SPLINE
SPL {X  -165.650, Y  +503.302, Z    +0.000, E1   +50.402, E3 +249333.532}
SPL {X  -165.650, Y  +495.166, Z    +0.000, E1   +51.070, E3 +249343.108}
SPL {X  -165.650, Y  +485.807, Z    +0.000, E1   +51.973, E3 +249352.841}
SPL {X  -165.650, Y  +478.030, Z    +0.000, E1   +52.389, E3 +249362.648}
SPL {X  -165.650, Y  +467.527, Z    +0.000, E1   +53.334, E3 +249373.142}
SPL {X  -165.650, Y  +457.379, Z    +0.000, E1   +53.935, E3 +249384.686}
SPL {X  -165.650, Y  +444.120, Z    +0.000, E1   +54.815, E3 +249398.731}
SPL {X  -165.650, Y  +431.771, Z    +0.000, E1   +55.549, E3 +249411.561}
SPL {X  -165.650, Y  +420.799, Z    +0.000, E1   +56.452, E3 +249420.947}
SPL {X  -165.650, Y  +409.731, Z    +0.000, E1   +57.273, E3 +249430.435}
SPL {X  -165.650, Y  +399.687, Z    +0.000, E1   +57.433, E3 +249442.620}
SPL {X  -165.650, Y  +388.492, Z    +0.000, E1   +57.709, E3 +249455.333}
SPL {X  -165.650, Y  +379.894, Z    +0.000, E1   +57.709, E3 +249466.436}
SPL {X  -165.538, Y  +372.423, Z    +0.000, E1   +57.528, E3 +249477.309}
SPL {X  -164.865, Y  +362.388, Z    +0.000, E1   +57.628, E3 +249489.696}
SPL {X  -163.867, Y  +354.258, Z    +0.000, E1   +57.359, E3 +249501.913}
SPL {X  -162.678, Y  +347.264, Z    +0.000, E1   +57.150, E3 +249512.254}
SPL {X  -161.618, Y  +342.173, Z    +0.000, E1   +56.783, E3 +249521.140}
SPL {X  -159.878, Y  +335.155, Z    +0.000, E1   +56.685, E3 +249530.943}
SPL {X  -158.009, Y  +328.771, Z    +0.000, E1   +56.325, E3 +249541.303}
SPL {X  -156.065, Y  +322.971, Z    +0.000, E1   +56.177, E3 +249549.647}
SPL {X  -154.487, Y  +318.719, Z    +0.000, E1   +55.733, E3 +249557.655}
SPL {X  -151.902, Y  +312.426, Z    +0.000, E1   +55.494, E3 +249567.130}
SPL {X  -149.742, Y  +307.668, Z    +0.000, E1   +54.896, E3 +249576.343}
SPL {X  -146.487, Y  +301.160, Z    +0.000, E1   +54.808, E3 +249585.205}
SPL {X  -133.590, Y  +280.553, Z    +0.000, E1   +59.642, E3 +249586.162}
SPL {X  -112.638, Y  +257.040, Z    +0.000, E1   +51.417, E3 +249689.546}
ENDSPLINE

SPLINE
SPL {X  -115.209, Y  +259.476, Z    +0.000, E1   +49.595, E3 +249722.816}
SPL {X  -147.344, Y  +302.806, Z    +0.000, E1   +40.158, E3 +249812.278}
SPL {X  -160.798, Y  +338.700, Z    +0.000, E1   +25.294, E3 +249811.760}
SPL {X  -163.893, Y  +354.439, Z    +0.000, E1   +16.805, E3 +249806.234}
SPL {X  -165.158, Y  +365.746, Z    +0.000, E1   +10.198, E3 +249804.177}
SPL {X  -165.580, Y  +373.688, Z    +0.000, E1    +5.094, E3 +249803.914}
SPL {X  -165.650, Y  +379.719, Z    +0.000, E1    +0.894, E3 +249803.344}
SPL {X  -165.650, Y  +383.454, Z    +0.000, E1    -2.667, E3 +249802.412}
SPL {X  -165.650, Y  +387.779, Z    +0.000, E1    -8.159, E3 +249802.085}
SPL {X  -165.650, Y  +392.511, Z    +0.000, E1   -14.940, E3 +249800.576}
SPL {X  -165.650, Y  +401.614, Z    +0.000, E1   -27.619, E3 +249801.318}
SPL {X  -165.650, Y  +418.105, Z    +0.000, E1   -49.413, E3 +249796.726}
SPL {X  -165.650, Y  +465.736, Z    +0.000, E1   -65.678, E3 +249810.468}
SPL {X  -165.650, Y  +519.483, Z    +0.000, E1   -68.357, E3 +249836.653}
SPL {X  -165.650, Y  +548.869, Z    +0.000, E1   -62.199, E3 +249892.346}
ENDSPLINE

SPLINE
SPL {X  -165.650, Y  +530.735, Z    +0.000, E1   -57.778, E3 +249900.769}
ENDSPLINE

SPLINE
SPL {X  -165.650, Y  +536.777, Z    +0.000, E1   -57.774, E3 +249908.646}
SPL {X  -165.650, Y  +545.905, Z    +0.000, E1   -57.853, E3 +249919.934}
SPL {X  -165.650, Y  +553.630, Z    +0.000, E1   -57.616, E3 +249931.384}
SPL {X  -165.650, Y  +563.473, Z    +0.000, E1   -57.690, E3 +249943.748}
SPL {X  -165.650, Y  +573.011, Z    +0.000, E1   -57.610, E3 +249956.539}
SPL {X  -165.650, Y  +581.530, Z    +0.000, E1   -57.678, E3 +249967.137}
SPL {X  -165.650, Y  +589.475, Z    +0.000, E1   -57.572, E3 +249978.124}
SPL {X  -165.650, Y  +599.695, Z    +0.000, E1   -57.964, E3 +249988.740}
SPL {X  -165.650, Y  +606.915, Z    +0.000, E1   -57.651, E3 +250000.097}
SPL {X  -165.650, Y  +614.927, Z    +0.000, E1   -57.517, E3 +250011.367}
SPL {X  -165.650, Y  +624.337, Z    +0.000, E1   -57.671, E3 +250022.593}
SPL {X  -165.650, Y  +634.236, Z    +0.000, E1   -57.671, E3 +250035.443}
SPL {X  -165.650, Y  +647.519, Z    +0.000, E1   -57.817, E3 +250051.770}
SPL {X  -165.650, Y  +657.986, Z    +0.000, E1   -57.646, E3 +250066.206}
SPL {X  -165.650, Y  +667.585, Z    +0.000, E1   -57.803, E3 +250077.602}
SPL {X  -165.634, Y  +677.794, Z    +0.000, E1   -57.650, E3 +250091.904}
SPL {X  -165.167, Y  +688.139, Z    +0.000, E1   -57.463, E3 +250106.483}
SPL {X  -164.323, Y  +696.426, Z    +0.000, E1   -57.565, E3 +250116.470}
SPL {X  -163.313, Y  +703.224, Z    +0.000, E1   -57.403, E3 +250126.364}
SPL {X  -161.906, Y  +710.520, Z    +0.000, E1   -57.149, E3 +250137.315}
SPL {X  -160.577, Y  +716.182, Z    +0.000, E1   -56.676, E3 +250147.576}
SPL {X  -158.520, Y  +723.576, Z    +0.000, E1   -56.758, E3 +250156.621}
SPL {X  -156.858, Y  +728.749, Z    +0.000, E1   -56.333, E3 +250165.763}
SPL {X  -155.155, Y  +733.525, Z    +0.000, E1   -55.869, E3 +250174.540}
SPL {X  -153.442, Y  +737.914, Z    +0.000, E1   -55.562, E3 +250181.945}
SPL {X  -150.574, Y  +744.547, Z    +0.000, E1   -55.310, E3 +250191.927}
SPL {X  -147.713, Y  +750.471, Z    +0.000, E1   -54.514, E3 +250203.590}
SPL {X  -139.786, Y  +764.381, Z    +0.000, E1   -57.209, E3 +250207.778}
SPL {X  -110.324, Y  +799.066, Z    +0.000, E1   -54.396, E3 +250276.352}
SPL {X  -100.308, Y  +807.326, Z    +0.000, E1   -52.880, E3 +250320.919}
ENDSPLINE

SPLINE
SPL {X  -108.196, Y  +800.934, Z    +0.000, E1   -52.068, E3 +250413.246}
SPL {X  -144.673, Y  +756.182, Z    +0.000, E1   -41.752, E3 +250431.325}
SPL {X  -160.601, Y  +716.087, Z    +0.000, E1   -25.730, E3 +250430.952}
SPL {X  -164.850, Y  +691.761, Z    +0.000, E1   -12.424, E3 +250428.220}
SPL {X  -165.596, Y  +679.730, Z    +0.000, E1    -4.777, E3 +250427.093}
SPL {X  -165.650, Y  +674.376, Z    +0.000, E1    -0.866, E3 +250427.009}
SPL {X  -165.650, Y  +672.384, Z    +0.000, E1    +0.908, E3 +250425.890}
SPL {X  -165.650, Y  +669.093, Z    +0.000, E1    +4.549, E3 +250425.741}
SPL {X  -165.650, Y  +663.273, Z    +0.000, E1   +12.448, E3 +250424.978}
SPL {X  -165.650, Y  +654.885, Z    +0.000, E1   +25.204, E3 +250423.530}
SPL {X  -165.650, Y  +641.882, Z    +0.000, E1   +46.566, E3 +250416.401}
SPL {X  -165.650, Y  +630.946, Z    +0.000, E1   +55.779, E3 +250417.076}
SPL {X  -165.650, Y  +590.135, Z    +0.000, E1   +59.110, E3 +250449.696}
SPL {X  -165.650, Y  +491.251, Z    +0.000, E1   +65.373, E3 +250509.125}
ENDSPLINE

SPLINE
SPL {X  -165.650, Y  +517.534, Z    +0.000, E1   +59.090, E3 +250523.722}
ENDSPLINE

SPLINE
SPL {X  -165.650, Y  +515.821, Z    +0.000, E1   +58.153, E3 +250532.170}
SPL {X  -165.650, Y  +506.715, Z    +0.000, E1   +58.090, E3 +250544.258}
SPL {X  -165.650, Y  +496.085, Z    +0.000, E1   +57.984, E3 +250558.506}
SPL {X  -165.650, Y  +485.167, Z    +0.000, E1   +58.003, E3 +250572.338}
ENDSPLINE

SPLINE
SPL {X  -165.650, Y  +505.180, Z    +0.000, E1   +52.333, E3 +250579.090}
SPL {X  -165.650, Y  +506.534, Z    +0.000, E1   +50.148, E3 +250590.549}
ENDSPLINE

SPLINE
SPL {X  -165.650, Y  +495.166, Z    +0.000, E1   +51.070, E3 +250603.978}
SPL {X  -165.650, Y  +485.807, Z    +0.000, E1   +51.973, E3 +250613.711}
SPL {X  -165.650, Y  +478.030, Z    +0.000, E1   +52.389, E3 +250623.517}
SPL {X  -165.650, Y  +467.527, Z    +0.000, E1   +53.334, E3 +250634.012}
SPL {X  -165.650, Y  +453.744, Z    +0.000, E1   +54.190, E3 +250649.492}
SPL {X  -165.650, Y  +440.843, Z    +0.000, E1   +55.023, E3 +250662.913}
SPL {X  -165.650, Y  +431.771, Z    +0.000, E1   +55.549, E3 +250672.431}
SPL {X  -165.650, Y  +420.799, Z    +0.000, E1   +56.452, E3 +250681.816}
SPL {X  -165.650, Y  +409.731, Z    +0.000, E1   +57.273, E3 +250691.305}
SPL {X  -165.650, Y  +399.687, Z    +0.000, E1   +57.433, E3 +250703.489}
SPL {X  -165.650, Y  +388.492, Z    +0.000, E1   +57.709, E3 +250716.202}
SPL {X  -165.650, Y  +379.894, Z    +0.000, E1   +57.709, E3 +250727.306}
SPL {X  -165.399, Y  +369.388, Z    +0.000, E1   +57.657, E3 +250741.400}
SPL {X  -164.717, Y  +360.945, Z    +0.000, E1   +57.468, E3 +250753.338}
SPL {X  -163.867, Y  +354.258, Z    +0.000, E1   +57.359, E3 +250762.782}
SPL {X  -162.678, Y  +347.264, Z    +0.000, E1   +57.150, E3 +250773.124}
SPL {X  -161.618, Y  +342.173, Z    +0.000, E1   +56.783, E3 +250782.009}
SPL {X  -159.878, Y  +335.155, Z    +0.000, E1   +56.685, E3 +250791.813}
SPL {X  -158.009, Y  +328.771, Z    +0.000, E1   +56.325, E3 +250802.172}
SPL {X  -156.065, Y  +322.971, Z    +0.000, E1   +56.177, E3 +250810.516}
SPL {X  -153.731, Y  +316.803, Z    +0.000, E1   +55.737, E3 +250821.093}
SPL {X  -150.320, Y  +308.902, Z    +0.000, E1   +55.085, E3 +250834.789}
SPL {X  -147.957, Y  +304.011, Z    +0.000, E1   +54.431, E3 +250844.251}
SPL {X  -144.791, Y  +298.030, Z    +0.000, E1   +55.214, E3 +250848.109}
SPL {X  -133.590, Y  +280.553, Z    +0.000, E1   +59.642, E3 +250847.032}
SPL {X  -112.638, Y  +257.040, Z    +0.000, E1   +51.417, E3 +250950.415}
ENDSPLINE

SPLINE
SPL {X  -115.209, Y  +259.476, Z    +0.000, E1   +49.595, E3 +250983.685}
SPL {X  -147.344, Y  +302.806, Z    +0.000, E1   +40.158, E3 +251073.148}
SPL {X  -160.798, Y  +338.700, Z    +0.000, E1   +25.294, E3 +251072.630}
SPL {X  -163.893, Y  +354.439, Z    +0.000, E1   +16.805, E3 +251067.104}
SPL {X  -165.158, Y  +365.746, Z    +0.000, E1   +10.198, E3 +251065.046}
SPL {X  -165.580, Y  +373.688, Z    +0.000, E1    +5.094, E3 +251064.783}
SPL {X  -165.650, Y  +379.719, Z    +0.000, E1    +0.894, E3 +251064.213}
SPL {X  -165.650, Y  +383.454, Z    +0.000, E1    -2.667, E3 +251063.281}
SPL {X  -165.650, Y  +387.779, Z    +0.000, E1    -8.159, E3 +251062.955}
SPL {X  -165.650, Y  +392.511, Z    +0.000, E1   -14.940, E3 +251061.446}
SPL {X  -165.650, Y  +401.614, Z    +0.000, E1   -27.619, E3 +251062.187}
SPL {X  -165.650, Y  +418.105, Z    +0.000, E1   -49.413, E3 +251057.595}
SPL {X  -165.650, Y  +465.736, Z    +0.000, E1   -65.678, E3 +251071.338}
SPL {X  -165.650, Y  +519.483, Z    +0.000, E1   -68.357, E3 +251097.523}
SPL {X  -165.650, Y  +548.869, Z    +0.000, E1   -62.199, E3 +251153.215}
ENDSPLINE

SPLINE
SPL {X  -165.650, Y  +534.780, Z    +0.000, E1   -57.803, E3 +251166.864}
ENDSPLINE

SPLINE
SPL {X  -165.650, Y  +545.905, Z    +0.000, E1   -57.853, E3 +251180.804}
SPL {X  -165.650, Y  +555.746, Z    +0.000, E1   -57.571, E3 +251195.442}
SPL {X  -165.650, Y  +566.557, Z    +0.000, E1   -57.834, E3 +251207.569}
SPL {X  -165.650, Y  +573.011, Z    +0.000, E1   -57.610, E3 +251217.409}
SPL {X  -165.650, Y  +581.530, Z    +0.000, E1   -57.678, E3 +251228.007}
SPL {X  -165.650, Y  +589.475, Z    +0.000, E1   -57.572, E3 +251238.994}
SPL {X  -165.650, Y  +599.695, Z    +0.000, E1   -57.964, E3 +251249.610}
SPL {X  -165.650, Y  +606.915, Z    +0.000, E1   -57.651, E3 +251260.967}
SPL {X  -165.650, Y  +614.927, Z    +0.000, E1   -57.517, E3 +251272.236}
SPL {X  -165.650, Y  +624.337, Z    +0.000, E1   -57.671, E3 +251283.462}
SPL {X  -165.650, Y  +634.236, Z    +0.000, E1   -57.671, E3 +251296.313}
SPL {X  -165.650, Y  +647.519, Z    +0.000, E1   -57.817, E3 +251312.640}
SPL {X  -165.650, Y  +657.986, Z    +0.000, E1   -57.646, E3 +251327.075}
SPL {X  -165.650, Y  +667.585, Z    +0.000, E1   -57.803, E3 +251338.471}
SPL {X  -165.634, Y  +677.794, Z    +0.000, E1   -57.650, E3 +251352.773}
SPL {X  -165.167, Y  +688.139, Z    +0.000, E1   -57.463, E3 +251367.353}
SPL {X  -164.009, Y  +698.761, Z    +0.000, E1   -57.613, E3 +251380.126}
SPL {X  -162.382, Y  +708.242, Z    +0.000, E1   -57.205, E3 +251395.052}
SPL {X  -160.577, Y  +716.182, Z    +0.000, E1   -56.676, E3 +251408.446}
SPL {X  -158.520, Y  +723.576, Z    +0.000, E1   -56.758, E3 +251417.490}
SPL {X  -156.858, Y  +728.749, Z    +0.000, E1   -56.333, E3 +251426.633}
SPL {X  -155.155, Y  +733.525, Z    +0.000, E1   -55.869, E3 +251435.410}
SPL {X  -152.530, Y  +740.111, Z    +0.000, E1   -55.545, E3 +251445.886}
SPL {X  -149.838, Y  +746.130, Z    +0.000, E1   -55.135, E3 +251455.606}
SPL {X  -147.713, Y  +750.471, Z    +0.000, E1   -54.514, E3 +251464.459}
SPL {X  -139.786, Y  +764.381, Z    +0.000, E1   -57.209, E3 +251468.648}
SPL {X  -110.324, Y  +799.066, Z    +0.000, E1   -54.396, E3 +251537.222}
SPL {X  -100.308, Y  +807.326, Z    +0.000, E1   -52.880, E3 +251581.789}
ENDSPLINE

SPLINE
SPL {X  -108.196, Y  +800.934, Z    +0.000, E1   -52.068, E3 +251674.115}
SPL {X  -147.753, Y  +750.393, Z    +0.000, E1   -39.863, E3 +251692.338}
SPL {X  -161.414, Y  +712.720, Z    +0.000, E1   -24.024, E3 +251691.680}
SPL {X  -164.278, Y  +696.774, Z    +0.000, E1   -15.225, E3 +251686.292}
SPL {X  -165.078, Y  +689.251, Z    +0.000, E1   -10.876, E3 +251690.444}
SPL {X  -165.596, Y  +679.730, Z    +0.000, E1    -4.777, E3 +251687.963}
SPL {X  -165.650, Y  +674.376, Z    +0.000, E1    -0.866, E3 +251687.878}
SPL {X  -165.650, Y  +672.384, Z    +0.000, E1    +0.908, E3 +251686.759}
SPL {X  -165.650, Y  +669.093, Z    +0.000, E1    +4.549, E3 +251686.611}
SPL {X  -165.650, Y  +663.273, Z    +0.000, E1   +12.448, E3 +251685.848}
SPL {X  -165.650, Y  +657.199, Z    +0.000, E1   +21.720, E3 +251685.117}
SPL {X  -165.650, Y  +652.963, Z    +0.000, E1   +28.395, E3 +251683.803}
SPL {X  -165.650, Y  +641.882, Z    +0.000, E1   +46.566, E3 +251677.271}
SPL {X  -165.650, Y  +630.946, Z    +0.000, E1   +55.779, E3 +251677.946}
SPL {X  -165.650, Y  +590.135, Z    +0.000, E1   +59.110, E3 +251710.565}
SPL {X  -165.650, Y  +491.251, Z    +0.000, E1   +65.373, E3 +251769.994}
ENDSPLINE

SPLINE
SPL {X  -165.650, Y  +516.236, Z    +0.000, E1   +58.457, E3 +251790.675}
ENDSPLINE

SPLINE
SPL {X  -165.650, Y  +506.715, Z    +0.000, E1   +58.090, E3 +251805.128}
SPL {X  -165.650, Y  +496.085, Z    +0.000, E1   +57.984, E3 +251819.375}
SPL {X  -165.650, Y  +485.167, Z    +0.000, E1   +58.003, E3 +251833.207}
ENDSPLINE

SPLINE
SPL {X  -165.650, Y  +505.180, Z    +0.000, E1   +52.333, E3 +251839.959}
SPL {X  -165.650, Y  +506.534, Z    +0.000, E1   +50.148, E3 +251851.419}
ENDSPLINE

SPLINE
SPL {X  -165.650, Y  +495.166, Z    +0.000, E1   +51.070, E3 +251864.847}
SPL {X  -165.650, Y  +485.807, Z    +0.000, E1   +51.973, E3 +251874.580}
SPL {X  -165.650, Y  +475.672, Z    +0.000, E1   +52.573, E3 +251887.034}
SPL {X  -165.650, Y  +459.814, Z    +0.000, E1   +53.888, E3 +251903.223}
SPL {X  -165.650, Y  +448.876, Z    +0.000, E1   +54.452, E3 +251915.718}
SPL {X  -165.650, Y  +440.843, Z    +0.000, E1   +55.023, E3 +251923.782}
SPL {X  -165.650, Y  +431.771, Z    +0.000, E1   +55.549, E3 +251933.300}
SPL {X  -165.650, Y  +420.799, Z    +0.000, E1   +56.452, E3 +251942.686}
SPL {X  -165.650, Y  +406.746, Z    +0.000, E1   +57.489, E3 +251954.731}
SPL {X  -165.650, Y  +399.455, Z    +0.000, E1   +57.184, E3 +251966.153}
SPL {X  -165.650, Y  +388.492, Z    +0.000, E1   +57.709, E3 +251977.072}
SPL {X  -165.650, Y  +379.894, Z    +0.000, E1   +57.709, E3 +251988.176}
SPL {X  -165.399, Y  +369.388, Z    +0.000, E1   +57.657, E3 +252002.269}
SPL {X  -164.717, Y  +360.945, Z    +0.000, E1   +57.468, E3 +252014.207}
SPL {X  -163.867, Y  +354.258, Z    +0.000, E1   +57.359, E3 +252023.652}
SPL {X  -162.678, Y  +347.264, Z    +0.000, E1   +57.150, E3 +252033.993}
SPL {X  -160.825, Y  +338.812, Z    +0.000, E1   +56.892, E3 +252046.735}
SPL {X  -158.481, Y  +330.294, Z    +0.000, E1   +56.303, E3 +252061.254}
SPL {X  -156.065, Y  +322.971, Z    +0.000, E1   +56.177, E3 +252071.386}
SPL {X  -154.487, Y  +318.719, Z    +0.000, E1   +55.733, E3 +252079.395}
SPL {X  -151.902, Y  +312.426, Z    +0.000, E1   +55.494, E3 +252088.870}
SPL {X  -148.935, Y  +305.985, Z    +0.000, E1   +54.737, E3 +252101.246}
SPL {X  -144.791, Y  +298.030, Z    +0.000, E1   +55.214, E3 +252108.979}
SPL {X  -133.590, Y  +280.553, Z    +0.000, E1   +59.642, E3 +252107.901}
SPL {X  -112.638, Y  +257.040, Z    +0.000, E1   +51.417, E3 +252211.285}
ENDSPLINE

SPLINE
SPL {X  -115.209, Y  +259.476, Z    +0.000, E1   +49.595, E3 +252244.555}
SPL {X  -147.344, Y  +302.806, Z    +0.000, E1   +40.158, E3 +252334.017}
SPL {X  -160.798, Y  +338.700, Z    +0.000, E1   +25.294, E3 +252333.499}
SPL {X  -163.893, Y  +354.439, Z    +0.000, E1   +16.805, E3 +252327.973}
SPL {X  -165.158, Y  +365.746, Z    +0.000, E1   +10.198, E3 +252325.916}
SPL {X  -165.639, Y  +376.620, Z    +0.000, E1    +3.186, E3 +252325.716}
SPL {X  -165.650, Y  +380.533, Z    +0.000, E1    +0.120, E3 +252324.744}
SPL {X  -165.650, Y  +383.454, Z    +0.000, E1    -2.667, E3 +252324.151}
SPL {X  -165.650, Y  +388.792, Z    +0.000, E1    -9.482, E3 +252323.245}
SPL {X  -165.650, Y  +393.970, Z    +0.000, E1   -17.146, E3 +252322.402}
SPL {X  -165.650, Y  +401.614, Z    +0.000, E1   -27.619, E3 +252323.057}
SPL {X  -165.650, Y  +418.105, Z    +0.000, E1   -49.413, E3 +252318.465}
SPL {X  -165.650, Y  +465.736, Z    +0.000, E1   -65.678, E3 +252332.207}
SPL {X  -165.650, Y  +519.483, Z    +0.000, E1   -68.357, E3 +252358.392}
SPL {X  -165.650, Y  +548.869, Z    +0.000, E1   -62.199, E3 +252414.085}
ENDSPLINE

SPLINE
SPL {X  -165.650, Y  +534.780, Z    +0.000, E1   -57.803, E3 +252427.734}
ENDSPLINE

SPLINE
SPL {X  -165.650, Y  +545.905, Z    +0.000, E1   -57.853, E3 +252441.673}
SPL {X  -165.650, Y  +553.630, Z    +0.000, E1   -57.616, E3 +252453.123}
SPL {X  -165.650, Y  +563.473, Z    +0.000, E1   -57.690, E3 +252465.487}
SPL {X  -165.650, Y  +573.011, Z    +0.000, E1   -57.610, E3 +252478.278}
SPL {X  -165.650, Y  +581.530, Z    +0.000, E1   -57.678, E3 +252488.876}
SPL {X  -165.650, Y  +589.475, Z    +0.000, E1   -57.572, E3 +252499.863}
SPL {X  -165.650, Y  +599.695, Z    +0.000, E1   -57.964, E3 +252510.479}
SPL {X  -165.650, Y  +606.915, Z    +0.000, E1   -57.651, E3 +252521.836}
SPL {X  -165.650, Y  +614.927, Z    +0.000, E1   -57.517, E3 +252533.106}
SPL {X  -165.650, Y  +624.337, Z    +0.000, E1   -57.671, E3 +252544.332}
SPL {X  -165.650, Y  +634.236, Z    +0.000, E1   -57.671, E3 +252557.182}
SPL {X  -165.650, Y  +647.519, Z    +0.000, E1   -57.817, E3 +252573.509}
SPL {X  -165.650, Y  +657.986, Z    +0.000, E1   -57.646, E3 +252587.945}
SPL {X  -165.650, Y  +667.585, Z    +0.000, E1   -57.803, E3 +252599.341}
SPL {X  -165.634, Y  +677.794, Z    +0.000, E1   -57.650, E3 +252613.643}
SPL {X  -165.167, Y  +688.139, Z    +0.000, E1   -57.463, E3 +252628.222}
SPL {X  -164.009, Y  +698.761, Z    +0.000, E1   -57.613, E3 +252640.996}
SPL {X  -162.382, Y  +708.242, Z    +0.000, E1   -57.205, E3 +252655.921}
SPL {X  -160.577, Y  +716.182, Z    +0.000, E1   -56.676, E3 +252669.315}
SPL {X  -158.520, Y  +723.576, Z    +0.000, E1   -56.758, E3 +252678.360}
SPL {X  -156.858, Y  +728.749, Z    +0.000, E1   -56.333, E3 +252687.502}
SPL {X  -155.155, Y  +733.525, Z    +0.000, E1   -55.869, E3 +252696.279}
SPL {X  -153.442, Y  +737.914, Z    +0.000, E1   -55.562, E3 +252703.684}
SPL {X  -150.574, Y  +744.547, Z    +0.000, E1   -55.310, E3 +252713.666}
SPL {X  -147.713, Y  +750.471, Z    +0.000, E1   -54.514, E3 +252725.329}
SPL {X  -139.786, Y  +764.381, Z    +0.000, E1   -57.209, E3 +252729.517}
SPL {X  -110.324, Y  +799.066, Z    +0.000, E1   -54.396, E3 +252798.091}
SPL {X  -100.308, Y  +807.326, Z    +0.000, E1   -52.880, E3 +252842.658}
ENDSPLINE

SPLINE
SPL {X  -108.196, Y  +800.934, Z    +0.000, E1   -52.068, E3 +252934.985}
SPL {X  -144.673, Y  +756.182, Z    +0.000, E1   -41.752, E3 +252953.064}
SPL {X  -160.601, Y  +716.087, Z    +0.000, E1   -25.730, E3 +252952.691}
SPL {X  -164.850, Y  +691.761, Z    +0.000, E1   -12.424, E3 +252949.959}
SPL {X  -165.596, Y  +679.730, Z    +0.000, E1    -4.777, E3 +252948.832}
SPL {X  -165.650, Y  +674.376, Z    +0.000, E1    -0.866, E3 +252948.748}
SPL {X  -165.650, Y  +672.384, Z    +0.000, E1    +0.908, E3 +252947.629}
SPL {X  -165.650, Y  +669.093, Z    +0.000, E1    +4.549, E3 +252947.480}
SPL {X  -165.650, Y  +663.273, Z    +0.000, E1   +12.448, E3 +252946.717}
SPL {X  -165.650, Y  +654.885, Z    +0.000, E1   +25.204, E3 +252945.269}
SPL {X  -165.650, Y  +641.882, Z    +0.000, E1   +46.566, E3 +252938.140}
SPL {X  -165.650, Y  +630.946, Z    +0.000, E1   +55.779, E3 +252938.815}
SPL {X  -165.650, Y  +595.858, Z    +0.000, E1   +64.262, E3 +252953.696}
SPL {X  -165.650, Y  +589.368, Z    +0.000, E1   +58.232, E3 +252974.437}
SPL {X  -165.650, Y  +491.251, Z    +0.000, E1   +65.373, E3 +253030.864}
ENDSPLINE

SPLINE
SPL {X  -165.650, Y  +516.236, Z    +0.000, E1   +58.457, E3 +253051.545}
ENDSPLINE

SPLINE
SPL {X  -165.650, Y  +506.715, Z    +0.000, E1   +58.090, E3 +253065.998}
SPL {X  -165.650, Y  +496.085, Z    +0.000, E1   +57.984, E3 +253080.245}
SPL {X  -165.650, Y  +485.167, Z    +0.000, E1   +58.003, E3 +253094.077}
ENDSPLINE

SPLINE
SPL {X  -165.650, Y  +505.180, Z    +0.000, E1   +52.333, E3 +253100.829}
SPL {X  -165.650, Y  +506.534, Z    +0.000, E1   +50.148, E3 +253112.288}
ENDSPLINE

SPLINE
SPL {X  -165.650, Y  +495.166, Z    +0.000, E1   +51.070, E3 +253125.717}
SPL {X  -165.650, Y  +485.807, Z    +0.000, E1   +51.973, E3 +253135.450}
SPL {X  -165.650, Y  +475.672, Z    +0.000, E1   +52.573, E3 +253147.903}
SPL {X  -165.650, Y  +459.814, Z    +0.000, E1   +53.888, E3 +253164.093}
SPL {X  -165.650, Y  +448.876, Z    +0.000, E1   +54.452, E3 +253176.588}
SPL {X  -165.650, Y  +440.843, Z    +0.000, E1   +55.023, E3 +253184.652}
SPL {X  -165.650, Y  +431.771, Z    +0.000, E1   +55.549, E3 +253194.170}
SPL {X  -165.650, Y  +420.799, Z    +0.000, E1   +56.452, E3 +253203.555}
SPL {X  -165.650, Y  +409.731, Z    +0.000, E1   +57.273, E3 +253213.044}
SPL {X  -165.650, Y  +399.687, Z    +0.000, E1   +57.433, E3 +253225.228}
SPL {X  -165.650, Y  +388.492, Z    +0.000, E1   +57.709, E3 +253237.941}
SPL {X  -165.650, Y  +379.894, Z    +0.000, E1   +57.709, E3 +253249.045}
SPL {X  -165.538, Y  +372.423, Z    +0.000, E1   +57.528, E3 +253259.918}
SPL {X  -164.865, Y  +362.388, Z    +0.000, E1   +57.628, E3 +253272.305}
SPL {X  -163.867, Y  +354.258, Z    +0.000, E1   +57.359, E3 +253284.521}
SPL {X  -162.678, Y  +347.264, Z    +0.000, E1   +57.150, E3 +253294.863}
SPL {X  -161.618, Y  +342.173, Z    +0.000, E1   +56.783, E3 +253303.748}
SPL {X  -159.878, Y  +335.155, Z    +0.000, E1   +56.685, E3 +253313.552}
SPL {X  -158.009, Y  +328.771, Z    +0.000, E1   +56.325, E3 +253323.912}
SPL {X  -156.065, Y  +322.971, Z    +0.000, E1   +56.177, E3 +253332.256}
SPL {X  -154.487, Y  +318.719, Z    +0.000, E1   +55.733, E3 +253340.264}
SPL {X  -151.902, Y  +312.426, Z    +0.000, E1   +55.494, E3 +253349.739}
SPL {X  -148.935, Y  +305.985, Z    +0.000, E1   +54.737, E3 +253362.116}
SPL {X  -144.791, Y  +298.030, Z    +0.000, E1   +55.214, E3 +253369.848}
SPL {X  -133.590, Y  +280.553, Z    +0.000, E1   +59.642, E3 +253368.771}
SPL {X  -112.638, Y  +257.040, Z    +0.000, E1   +51.417, E3 +253472.154}
ENDSPLINE

SPLINE
SPL {X  -115.209, Y  +259.476, Z    +0.000, E1   +49.595, E3 +253505.425}
SPL {X  -147.344, Y  +302.806, Z    +0.000, E1   +40.158, E3 +253594.887}
SPL {X  -160.798, Y  +338.700, Z    +0.000, E1   +25.294, E3 +253594.369}
SPL {X  -163.893, Y  +354.439, Z    +0.000, E1   +16.805, E3 +253588.843}
SPL {X  -165.158, Y  +365.746, Z    +0.000, E1   +10.198, E3 +253586.786}
SPL {X  -165.580, Y  +373.688, Z    +0.000, E1    +5.094, E3 +253586.523}
SPL {X  -165.650, Y  +378.140, Z    +0.000, E1    +1.996, E3 +253586.609}
SPL {X  -165.650, Y  +381.477, Z    +0.000, E1    -0.622, E3 +253585.396}
SPL {X  -165.650, Y  +384.861, Z    +0.000, E1    -4.465, E3 +253584.799}
SPL {X  -165.650, Y  +388.792, Z    +0.000, E1    -9.482, E3 +253584.115}
SPL {X  -165.650, Y  +393.970, Z    +0.000, E1   -17.146, E3 +253583.271}
SPL {X  -165.650, Y  +401.614, Z    +0.000, E1   -27.619, E3 +253583.926}
SPL {X  -165.650, Y  +418.105, Z    +0.000, E1   -49.413, E3 +253579.334}
SPL {X  -165.650, Y  +465.736, Z    +0.000, E1   -65.678, E3 +253593.077}
SPL {X  -165.650, Y  +519.483, Z    +0.000, E1   -68.357, E3 +253619.262}
SPL {X  -165.650, Y  +548.869, Z    +0.000, E1   -62.199, E3 +253674.954}
ENDSPLINE

SPLINE
SPL {X  -165.650, Y  +534.780, Z    +0.000, E1   -57.803, E3 +253688.604}
ENDSPLINE

SPLINE
SPL {X  -165.650, Y  +545.905, Z    +0.000, E1   -57.853, E3 +253702.543}
SPL {X  -165.650, Y  +553.630, Z    +0.000, E1   -57.616, E3 +253713.993}
SPL {X  -165.650, Y  +563.473, Z    +0.000, E1   -57.690, E3 +253726.357}
SPL {X  -165.650, Y  +573.011, Z    +0.000, E1   -57.610, E3 +253739.148}
SPL {X  -165.650, Y  +581.530, Z    +0.000, E1   -57.678, E3 +253749.746}
SPL {X  -165.650, Y  +589.475, Z    +0.000, E1   -57.572, E3 +253760.733}
SPL {X  -165.650, Y  +599.695, Z    +0.000, E1   -57.964, E3 +253771.349}
SPL {X  -165.650, Y  +606.915, Z    +0.000, E1   -57.651, E3 +253782.706}
SPL {X  -165.650, Y  +614.927, Z    +0.000, E1   -57.517, E3 +253793.975}
SPL {X  -165.650, Y  +624.337, Z    +0.000, E1   -57.671, E3 +253805.201}
SPL {X  -165.650, Y  +634.236, Z    +0.000, E1   -57.671, E3 +253818.052}
SPL {X  -165.650, Y  +647.519, Z    +0.000, E1   -57.817, E3 +253834.379}
SPL {X  -165.650, Y  +657.986, Z    +0.000, E1   -57.646, E3 +253848.814}
SPL {X  -165.650, Y  +667.585, Z    +0.000, E1   -57.803, E3 +253860.210}
SPL {X  -165.634, Y  +677.794, Z    +0.000, E1   -57.650, E3 +253874.512}
SPL {X  -165.167, Y  +688.139, Z    +0.000, E1   -57.463, E3 +253889.092}
SPL {X  -164.009, Y  +698.761, Z    +0.000, E1   -57.613, E3 +253901.865}
SPL {X  -162.382, Y  +708.242, Z    +0.000, E1   -57.205, E3 +253916.791}
SPL {X  -160.577, Y  +716.182, Z    +0.000, E1   -56.676, E3 +253930.185}
SPL {X  -158.520, Y  +723.576, Z    +0.000, E1   -56.758, E3 +253939.230}
SPL {X  -156.858, Y  +728.749, Z    +0.000, E1   -56.333, E3 +253948.372}
SPL {X  -155.155, Y  +733.525, Z    +0.000, E1   -55.869, E3 +253957.149}
SPL {X  -152.530, Y  +740.111, Z    +0.000, E1   -55.545, E3 +253967.625}
SPL {X  -149.838, Y  +746.130, Z    +0.000, E1   -55.135, E3 +253977.345}
SPL {X  -147.713, Y  +750.471, Z    +0.000, E1   -54.514, E3 +253986.199}
SPL {X  -139.786, Y  +764.381, Z    +0.000, E1   -57.209, E3 +253990.387}
SPL {X  -110.324, Y  +799.066, Z    +0.000, E1   -54.396, E3 +254058.961}
SPL {X  -100.308, Y  +807.326, Z    +0.000, E1   -52.880, E3 +254103.528}
ENDSPLINE

SPLINE
SPL {X  -108.196, Y  +800.934, Z    +0.000, E1   -52.068, E3 +254195.854}
SPL {X  -144.673, Y  +756.182, Z    +0.000, E1   -41.752, E3 +254213.933}
SPL {X  -160.601, Y  +716.087, Z    +0.000, E1   -25.730, E3 +254213.561}
SPL {X  -164.850, Y  +691.761, Z    +0.000, E1   -12.424, E3 +254210.828}
SPL {X  -165.596, Y  +679.730, Z    +0.000, E1    -4.777, E3 +254209.702}
SPL {X  -165.650, Y  +674.376, Z    +0.000, E1    -0.866, E3 +254209.617}
SPL {X  -165.650, Y  +672.384, Z    +0.000, E1    +0.908, E3 +254208.498}
SPL {X  -165.650, Y  +669.968, Z    +0.000, E1    +3.584, E3 +254208.314}
SPL {X  -165.650, Y  +666.667, Z    +0.000, E1    +7.761, E3 +254207.993}
SPL {X  -165.650, Y  +662.028, Z    +0.000, E1   +14.359, E3 +254207.624}
SPL {X  -165.650, Y  +654.885, Z    +0.000, E1   +25.204, E3 +254206.139}
SPL {X  -165.650, Y  +641.882, Z    +0.000, E1   +46.566, E3 +254199.010}
SPL {X  -165.650, Y  +630.946, Z    +0.000, E1   +55.779, E3 +254199.685}
SPL {X  -165.650, Y  +590.135, Z    +0.000, E1   +59.110, E3 +254232.304}
SPL {X  -165.650, Y  +491.251, Z    +0.000, E1   +65.373, E3 +254291.734}
ENDSPLINE

SPLINE
SPL {X  -165.650, Y  +516.236, Z    +0.000, E1   +58.457, E3 +254312.414}
ENDSPLINE

SPLINE
SPL {X  -165.650, Y  +506.715, Z    +0.000, E1   +58.090, E3 +254326.867}
SPL {X  -165.650, Y  +496.085, Z    +0.000, E1   +57.984, E3 +254341.115}
SPL {X  -165.650, Y  +485.167, Z    +0.000, E1   +58.003, E3 +254354.946}
ENDSPLINE

SPLINE
SPL {X  -165.650, Y  +505.180, Z    +0.000, E1   +52.333, E3 +254361.698}
SPL {X  -165.650, Y  +506.534, Z    +0.000, E1   +50.148, E3 +254373.158}
ENDSPLINE

SPLINE
SPL {X  -165.650, Y  +495.166, Z    +0.000, E1   +51.070, E3 +254386.586}
SPL {X  -165.650, Y  +485.807, Z    +0.000, E1   +51.973, E3 +254396.319}
SPL {X  -165.650, Y  +478.030, Z    +0.000, E1   +52.389, E3 +254406.126}
SPL {X  -165.650, Y  +467.527, Z    +0.000, E1   +53.334, E3 +254416.620}
SPL {X  -165.650, Y  +457.379, Z    +0.000, E1   +53.935, E3 +254428.164}
SPL {X  -165.650, Y  +444.120, Z    +0.000, E1   +54.815, E3 +254442.209}
SPL {X  -165.650, Y  +431.771, Z    +0.000, E1   +55.549, E3 +254455.039}
SPL {X  -165.650, Y  +420.799, Z    +0.000, E1   +56.452, E3 +254464.425}
SPL {X  -165.650, Y  +409.731, Z    +0.000, E1   +57.273, E3 +254473.913}
SPL {X  -165.650, Y  +399.687, Z    +0.000, E1   +57.433, E3 +254486.098}
SPL {X  -165.650, Y  +388.492, Z    +0.000, E1   +57.709, E3 +254498.811}
SPL {X  -165.650, Y  +379.894, Z    +0.000, E1   +57.709, E3 +254509.915}
SPL {X  -165.538, Y  +372.423, Z    +0.000, E1   +57.528, E3 +254520.788}
SPL {X  -164.865, Y  +362.388, Z    +0.000, E1   +57.628, E3 +254533.174}
SPL {X  -163.867, Y  +354.258, Z    +0.000, E1   +57.359, E3 +254545.391}
SPL {X  -162.678, Y  +347.264, Z    +0.000, E1   +57.150, E3 +254555.732}
SPL {X  -161.618, Y  +342.173, Z    +0.000, E1   +56.783, E3 +254564.618}
SPL {X  -159.878, Y  +335.155, Z    +0.000, E1   +56.685, E3 +254574.421}
SPL {X  -158.009, Y  +328.771, Z    +0.000, E1   +56.325, E3 +254584.781}
SPL {X  -156.065, Y  +322.971, Z    +0.000, E1   +56.177, E3 +254593.125}
SPL {X  -154.487, Y  +318.719, Z    +0.000, E1   +55.733, E3 +254601.134}
SPL {X  -151.902, Y  +312.426, Z    +0.000, E1   +55.494, E3 +254610.609}
SPL {X  -149.742, Y  +307.668, Z    +0.000, E1   +54.896, E3 +254619.821}
SPL {X  -146.487, Y  +301.160, Z    +0.000, E1   +54.808, E3 +254628.684}
SPL {X  -133.590, Y  +280.553, Z    +0.000, E1   +59.642, E3 +254629.641}
SPL {X  -112.638, Y  +257.040, Z    +0.000, E1   +51.417, E3 +254733.024}
ENDSPLINE

SPLINE
SPL {X  -115.209, Y  +259.476, Z    +0.000, E1   +49.595, E3 +254766.294}
SPL {X  -147.344, Y  +302.806, Z    +0.000, E1   +40.158, E3 +254855.756}
SPL {X  -160.798, Y  +338.700, Z    +0.000, E1   +25.294, E3 +254855.238}
SPL {X  -163.893, Y  +354.439, Z    +0.000, E1   +16.805, E3 +254849.712}
SPL {X  -165.158, Y  +365.746, Z    +0.000, E1   +10.198, E3 +254847.655}
SPL {X  -165.639, Y  +376.620, Z    +0.000, E1    +3.186, E3 +254847.455}
SPL {X  -165.650, Y  +381.477, Z    +0.000, E1    -0.622, E3 +254846.266}
SPL {X  -165.650, Y  +386.363, Z    +0.000, E1    -6.162, E3 +254845.614}
SPL {X  -165.650, Y  +392.511, Z    +0.000, E1   -14.940, E3 +254844.054}
SPL {X  -165.650, Y  +398.939, Z    +0.000, E1   -23.851, E3 +254845.439}
SPL {X  -165.650, Y  +404.249, Z    +0.000, E1   -31.650, E3 +254844.161}
SPL {X  -165.650, Y  +418.105, Z    +0.000, E1   -49.413, E3 +254840.204}
SPL {X  -165.650, Y  +465.736, Z    +0.000, E1   -65.678, E3 +254853.946}
SPL {X  -165.650, Y  +519.483, Z    +0.000, E1   -68.357, E3 +254880.131}
SPL {X  -165.650, Y  +548.869, Z    +0.000, E1   -62.199, E3 +254935.824}
ENDSPLINE

SPLINE
SPL {X  -165.650, Y  +530.735, Z    +0.000, E1   -57.778, E3 +254944.247}
ENDSPLINE

SPLINE
SPL {X  -165.650, Y  +536.777, Z    +0.000, E1   -57.774, E3 +254952.124}
SPL {X  -165.650, Y  +545.905, Z    +0.000, E1   -57.853, E3 +254963.413}
SPL {X  -165.650, Y  +553.630, Z    +0.000, E1   -57.616, E3 +254974.862}
SPL {X  -165.650, Y  +563.473, Z    +0.000, E1   -57.690, E3 +254987.226}
SPL {X  -165.650, Y  +573.011, Z    +0.000, E1   -57.610, E3 +255000.017}
SPL {X  -165.650, Y  +581.530, Z    +0.000, E1   -57.678, E3 +255010.615}
SPL {X  -165.650, Y  +589.475, Z    +0.000, E1   -57.572, E3 +255021.602}
SPL {X  -165.650, Y  +599.695, Z    +0.000, E1   -57.964, E3 +255032.218}
SPL {X  -165.650, Y  +606.915, Z    +0.000, E1   -57.651, E3 +255043.575}
SPL {X  -165.650, Y  +614.927, Z    +0.000, E1   -57.517, E3 +255054.845}
SPL {X  -165.650, Y  +624.337, Z    +0.000, E1   -57.671, E3 +255066.071}
SPL {X  -165.650, Y  +634.236, Z    +0.000, E1   -57.671, E3 +255078.921}
SPL {X  -165.650, Y  +647.519, Z    +0.000, E1   -57.817, E3 +255095.249}
SPL {X  -165.650, Y  +657.986, Z    +0.000, E1   -57.646, E3 +255109.684}
SPL {X  -165.650, Y  +667.585, Z    +0.000, E1   -57.803, E3 +255121.080}
SPL {X  -165.634, Y  +677.794, Z    +0.000, E1   -57.650, E3 +255135.382}
SPL {X  -165.167, Y  +688.139, Z    +0.000, E1   -57.463, E3 +255149.961}
SPL {X  -164.323, Y  +696.426, Z    +0.000, E1   -57.565, E3 +255159.948}
SPL {X  -163.313, Y  +703.224, Z    +0.000, E1   -57.403, E3 +255169.842}
SPL {X  -161.906, Y  +710.520, Z    +0.000, E1   -57.149, E3 +255180.793}
SPL {X  -160.577, Y  +716.182, Z    +0.000, E1   -56.676, E3 +255191.054}
SPL {X  -158.520, Y  +723.576, Z    +0.000, E1   -56.758, E3 +255200.099}
SPL {X  -156.858, Y  +728.749, Z    +0.000, E1   -56.333, E3 +255209.242}
SPL {X  -155.155, Y  +733.525, Z    +0.000, E1   -55.869, E3 +255218.018}
SPL {X  -153.442, Y  +737.914, Z    +0.000, E1   -55.562, E3 +255225.423}
SPL {X  -150.574, Y  +744.547, Z    +0.000, E1   -55.310, E3 +255235.405}
SPL {X  -147.713, Y  +750.471, Z    +0.000, E1   -54.514, E3 +255247.068}
SPL {X  -139.786, Y  +764.381, Z    +0.000, E1   -57.209, E3 +255251.256}
SPL {X  -110.324, Y  +799.066, Z    +0.000, E1   -54.396, E3 +255319.830}
SPL {X  -100.308, Y  +807.326, Z    +0.000, E1   -52.880, E3 +255364.398}
ENDSPLINE

SPLINE
SPL {X  -108.196, Y  +800.934, Z    +0.000, E1   -52.068, E3 +255456.724}
SPL {X  -144.673, Y  +756.182, Z    +0.000, E1   -41.752, E3 +255474.803}
SPL {X  -160.601, Y  +716.087, Z    +0.000, E1   -25.730, E3 +255474.430}
SPL {X  -164.850, Y  +691.761, Z    +0.000, E1   -12.424, E3 +255471.698}
SPL {X  -165.596, Y  +679.730, Z    +0.000, E1    -4.777, E3 +255470.572}
SPL {X  -165.650, Y  +674.376, Z    +0.000, E1    -0.866, E3 +255470.487}
SPL {X  -165.650, Y  +672.384, Z    +0.000, E1    +0.908, E3 +255469.368}
SPL {X  -165.650, Y  +669.093, Z    +0.000, E1    +4.549, E3 +255469.219}
SPL {X  -165.650, Y  +663.273, Z    +0.000, E1   +12.448, E3 +255468.457}
SPL {X  -165.650, Y  +654.885, Z    +0.000, E1   +25.204, E3 +255467.008}
SPL {X  -165.650, Y  +641.882, Z    +0.000, E1   +46.566, E3 +255459.880}
SPL {X  -165.650, Y  +630.946, Z    +0.000, E1   +55.779, E3 +255460.554}
SPL {X  -165.650, Y  +590.135, Z    +0.000, E1   +59.110, E3 +255493.174}
SPL {X  -165.650, Y  +491.251, Z    +0.000, E1   +65.373, E3 +255552.603}
ENDSPLINE

SPLINE
SPL {X  -165.650, Y  +517.534, Z    +0.000, E1   +59.090, E3 +255567.201}
ENDSPLINE

SPLINE
SPL {X  -165.650, Y  +515.821, Z    +0.000, E1   +58.153, E3 +255575.648}
SPL {X  -165.650, Y  +506.715, Z    +0.000, E1   +58.090, E3 +255587.737}
SPL {X  -165.650, Y  +496.085, Z    +0.000, E1   +57.984, E3 +255601.984}
SPL {X  -165.650, Y  +485.167, Z    +0.000, E1   +58.003, E3 +255615.816}
ENDSPLINE

SPLINE
SPL {X  -165.650, Y  +505.180, Z    +0.000, E1   +52.333, E3 +255622.568}
SPL {X  -165.650, Y  +506.534, Z    +0.000, E1   +50.148, E3 +255634.028}
ENDSPLINE

SPLINE
SPL {X  -165.650, Y  +495.166, Z    +0.000, E1   +51.070, E3 +255647.456}
SPL {X  -165.650, Y  +485.807, Z    +0.000, E1   +51.973, E3 +255657.189}
SPL {X  -165.650, Y  +478.030, Z    +0.000, E1   +52.389, E3 +255666.996}
SPL {X  -165.650, Y  +467.527, Z    +0.000, E1   +53.334, E3 +255677.490}
SPL {X  -165.650, Y  +453.744, Z    +0.000, E1   +54.190, E3 +255692.971}
SPL {X  -165.650, Y  +440.843, Z    +0.000, E1   +55.023, E3 +255706.391}
SPL {X  -165.650, Y  +431.771, Z    +0.000, E1   +55.549, E3 +255715.909}
SPL {X  -165.650, Y  +420.799, Z    +0.000, E1   +56.452, E3 +255725.295}
SPL {X  -165.650, Y  +409.731, Z    +0.000, E1   +57.273, E3 +255734.783}
SPL {X  -165.650, Y  +399.687, Z    +0.000, E1   +57.433, E3 +255746.967}
SPL {X  -165.650, Y  +388.492, Z    +0.000, E1   +57.709, E3 +255759.681}
SPL {X  -165.650, Y  +379.894, Z    +0.000, E1   +57.709, E3 +255770.784}
SPL {X  -165.399, Y  +369.388, Z    +0.000, E1   +57.657, E3 +255784.878}
SPL {X  -164.717, Y  +360.945, Z    +0.000, E1   +57.468, E3 +255796.816}
SPL {X  -163.867, Y  +354.258, Z    +0.000, E1   +57.359, E3 +255806.261}
SPL {X  -162.678, Y  +347.264, Z    +0.000, E1   +57.150, E3 +255816.602}
SPL {X  -161.618, Y  +342.173, Z    +0.000, E1   +56.783, E3 +255825.487}
SPL {X  -159.878, Y  +335.155, Z    +0.000, E1   +56.685, E3 +255835.291}
SPL {X  -158.009, Y  +328.771, Z    +0.000, E1   +56.325, E3 +255845.651}
SPL {X  -156.065, Y  +322.971, Z    +0.000, E1   +56.177, E3 +255853.995}
SPL {X  -153.731, Y  +316.803, Z    +0.000, E1   +55.737, E3 +255864.571}
SPL {X  -150.320, Y  +308.902, Z    +0.000, E1   +55.085, E3 +255878.267}
SPL {X  -147.957, Y  +304.011, Z    +0.000, E1   +54.431, E3 +255887.730}
SPL {X  -144.791, Y  +298.030, Z    +0.000, E1   +55.214, E3 +255891.587}
SPL {X  -133.590, Y  +280.553, Z    +0.000, E1   +59.642, E3 +255890.510}
SPL {X  -112.638, Y  +257.040, Z    +0.000, E1   +51.417, E3 +255993.893}
ENDSPLINE

SPLINE
SPL {X  -115.209, Y  +259.476, Z    +0.000, E1   +49.595, E3 +256027.164}
SPL {X  -147.344, Y  +302.806, Z    +0.000, E1   +40.158, E3 +256116.626}
SPL {X  -160.798, Y  +338.700, Z    +0.000, E1   +25.294, E3 +256116.108}
SPL {X  -163.893, Y  +354.439, Z    +0.000, E1   +16.805, E3 +256110.582}
SPL {X  -165.158, Y  +365.746, Z    +0.000, E1   +10.198, E3 +256108.525}
SPL {X  -165.580, Y  +373.688, Z    +0.000, E1    +5.094, E3 +256108.262}
SPL {X  -165.650, Y  +379.719, Z    +0.000, E1    +0.894, E3 +256107.692}
SPL {X  -165.650, Y  +383.454, Z    +0.000, E1    -2.667, E3 +256106.760}
SPL {X  -165.650, Y  +387.779, Z    +0.000, E1    -8.159, E3 +256106.433}
SPL {X  -165.650, Y  +392.511, Z    +0.000, E1   -14.940, E3 +256104.924}
SPL {X  -165.650, Y  +401.614, Z    +0.000, E1   -27.619, E3 +256105.666}
SPL {X  -165.650, Y  +418.105, Z    +0.000, E1   -49.413, E3 +256101.073}
SPL {X  -165.650, Y  +465.736, Z    +0.000, E1   -65.678, E3 +256114.816}
SPL {X  -165.650, Y  +519.483, Z    +0.000, E1   -68.357, E3 +256141.001}
SPL {X  -165.650, Y  +548.869, Z    +0.000, E1   -62.199, E3 +256196.693}
ENDSPLINE

SPLINE
SPL {X  -165.650, Y  +534.780, Z    +0.000, E1   -57.803, E3 +256210.343}
ENDSPLINE

SPLINE
SPL {X  -165.650, Y  +545.905, Z    +0.000, E1   -57.853, E3 +256224.282}
SPL {X  -165.650, Y  +555.746, Z    +0.000, E1   -57.571, E3 +256238.920}
SPL {X  -165.650, Y  +566.557, Z    +0.000, E1   -57.834, E3 +256251.048}
SPL {X  -165.650, Y  +573.011, Z    +0.000, E1   -57.610, E3 +256260.887}
SPL {X  -165.650, Y  +581.530, Z    +0.000, E1   -57.678, E3 +256271.485}
SPL {X  -165.650, Y  +589.475, Z    +0.000, E1   -57.572, E3 +256282.472}
SPL {X  -165.650, Y  +599.695, Z    +0.000, E1   -57.964, E3 +256293.088}
SPL {X  -165.650, Y  +606.915, Z    +0.000, E1   -57.651, E3 +256304.445}
SPL {X  -165.650, Y  +614.927, Z    +0.000, E1   -57.517, E3 +256315.715}
SPL {X  -165.650, Y  +624.337, Z    +0.000, E1   -57.671, E3 +256326.940}
SPL {X  -165.650, Y  +634.236, Z    +0.000, E1   -57.671, E3 +256339.791}
SPL {X  -165.650, Y  +647.519, Z    +0.000, E1   -57.817, E3 +256356.118}
SPL {X  -165.650, Y  +657.986, Z    +0.000, E1   -57.646, E3 +256370.554}
SPL {X  -165.650, Y  +667.585, Z    +0.000, E1   -57.803, E3 +256381.949}
SPL {X  -165.634, Y  +677.794, Z    +0.000, E1   -57.650, E3 +256396.252}
SPL {X  -165.167, Y  +688.139, Z    +0.000, E1   -57.463, E3 +256410.831}
SPL {X  -164.009, Y  +698.761, Z    +0.000, E1   -57.613, E3 +256423.604}
SPL {X  -162.382, Y  +708.242, Z    +0.000, E1   -57.205, E3 +256438.530}
SPL {X  -160.577, Y  +716.182, Z    +0.000, E1   -56.676, E3 +256451.924}
SPL {X  -158.520, Y  +723.576, Z    +0.000, E1   -56.758, E3 +256460.969}
SPL {X  -156.858, Y  +728.749, Z    +0.000, E1   -56.333, E3 +256470.111}
SPL {X  -155.155, Y  +733.525, Z    +0.000, E1   -55.869, E3 +256478.888}
SPL {X  -152.530, Y  +740.111, Z    +0.000, E1   -55.545, E3 +256489.364}
SPL {X  -149.838, Y  +746.130, Z    +0.000, E1   -55.135, E3 +256499.084}
SPL {X  -147.713, Y  +750.471, Z    +0.000, E1   -54.514, E3 +256507.938}
SPL {X  -139.786, Y  +764.381, Z    +0.000, E1   -57.209, E3 +256512.126}
SPL {X  -110.324, Y  +799.066, Z    +0.000, E1   -54.396, E3 +256580.700}
SPL {X  -100.308, Y  +807.326, Z    +0.000, E1   -52.880, E3 +256625.267}
ENDSPLINE

SPLINE
SPL {X  -108.196, Y  +800.934, Z    +0.000, E1   -52.068, E3 +256717.594}
SPL {X  -147.753, Y  +750.393, Z    +0.000, E1   -39.863, E3 +256735.816}
SPL {X  -161.414, Y  +712.720, Z    +0.000, E1   -24.024, E3 +256735.158}
SPL {X  -164.278, Y  +696.774, Z    +0.000, E1   -15.225, E3 +256729.770}
SPL {X  -165.078, Y  +689.251, Z    +0.000, E1   -10.876, E3 +256733.922}
SPL {X  -165.596, Y  +679.730, Z    +0.000, E1    -4.777, E3 +256731.441}
SPL {X  -165.650, Y  +674.376, Z    +0.000, E1    -0.866, E3 +256731.357}
SPL {X  -165.650, Y  +672.384, Z    +0.000, E1    +0.908, E3 +256730.238}
SPL {X  -165.650, Y  +669.093, Z    +0.000, E1    +4.549, E3 +256730.089}
SPL {X  -165.650, Y  +663.273, Z    +0.000, E1   +12.448, E3 +256729.326}
SPL {X  -165.650, Y  +657.199, Z    +0.000, E1   +21.720, E3 +256728.595}
SPL {X  -165.650, Y  +652.963, Z    +0.000, E1   +28.395, E3 +256727.281}
SPL {X  -165.650, Y  +641.882, Z    +0.000, E1   +46.566, E3 +256720.749}
SPL {X  -165.650, Y  +630.946, Z    +0.000, E1   +55.779, E3 +256721.424}
SPL {X  -165.650, Y  +590.135, Z    +0.000, E1   +59.110, E3 +256754.043}
SPL {X  -165.650, Y  +491.251, Z    +0.000, E1   +65.373, E3 +256813.473}
ENDSPLINE

SPLINE
SPL {X  -165.650, Y  +516.236, Z    +0.000, E1   +58.457, E3 +256834.153}
ENDSPLINE

SPLINE
SPL {X  -165.650, Y  +506.715, Z    +0.000, E1   +58.090, E3 +256848.606}
SPL {X  -165.650, Y  +496.085, Z    +0.000, E1   +57.984, E3 +256862.854}
SPL {X  -165.650, Y  +485.167, Z    +0.000, E1   +58.003, E3 +256876.685}
ENDSPLINE

SPLINE
SPL {X  -165.650, Y  +505.180, Z    +0.000, E1   +52.333, E3 +256883.438}
SPL {X  -165.650, Y  +506.534, Z    +0.000, E1   +50.148, E3 +256894.897}
ENDSPLINE

SPLINE
SPL {X  -165.650, Y  +495.166, Z    +0.000, E1   +51.070, E3 +256908.326}
SPL {X  -165.650, Y  +485.807, Z    +0.000, E1   +51.973, E3 +256918.058}
SPL {X  -165.650, Y  +475.672, Z    +0.000, E1   +52.573, E3 +256930.512}
SPL {X  -165.650, Y  +459.814, Z    +0.000, E1   +53.888, E3 +256946.701}
SPL {X  -165.650, Y  +448.876, Z    +0.000, E1   +54.452, E3 +256959.196}
SPL {X  -165.650, Y  +440.843, Z    +0.000, E1   +55.023, E3 +256967.261}
SPL {X  -165.650, Y  +431.771, Z    +0.000, E1   +55.549, E3 +256976.778}
SPL {X  -165.650, Y  +420.799, Z    +0.000, E1   +56.452, E3 +256986.164}
SPL {X  -165.650, Y  +406.746, Z    +0.000, E1   +57.489, E3 +256998.209}
SPL {X  -165.650, Y  +399.455, Z    +0.000, E1   +57.184, E3 +257009.631}
SPL {X  -165.650, Y  +388.492, Z    +0.000, E1   +57.709, E3 +257020.550}
SPL {X  -165.650, Y  +379.894, Z    +0.000, E1   +57.709, E3 +257031.654}
SPL {X  -165.399, Y  +369.388, Z    +0.000, E1   +57.657, E3 +257045.748}
SPL {X  -164.717, Y  +360.945, Z    +0.000, E1   +57.468, E3 +257057.686}
SPL {X  -163.867, Y  +354.258, Z    +0.000, E1   +57.359, E3 +257067.130}
SPL {X  -162.678, Y  +347.264, Z    +0.000, E1   +57.150, E3 +257077.471}
SPL {X  -160.825, Y  +338.812, Z    +0.000, E1   +56.892, E3 +257090.214}
SPL {X  -158.481, Y  +330.294, Z    +0.000, E1   +56.303, E3 +257104.732}
SPL {X  -156.065, Y  +322.971, Z    +0.000, E1   +56.177, E3 +257114.864}
SPL {X  -154.487, Y  +318.719, Z    +0.000, E1   +55.733, E3 +257122.873}
SPL {X  -151.902, Y  +312.426, Z    +0.000, E1   +55.494, E3 +257132.348}
SPL {X  -148.935, Y  +305.985, Z    +0.000, E1   +54.737, E3 +257144.725}
SPL {X  -144.791, Y  +298.030, Z    +0.000, E1   +55.214, E3 +257152.457}
SPL {X  -133.590, Y  +280.553, Z    +0.000, E1   +59.642, E3 +257151.380}
SPL {X  -112.638, Y  +257.040, Z    +0.000, E1   +51.417, E3 +257254.763}
ENDSPLINE

SPLINE
SPL {X  -115.209, Y  +259.476, Z    +0.000, E1   +49.595, E3 +257288.033}
SPL {X  -147.344, Y  +302.806, Z    +0.000, E1   +40.158, E3 +257377.495}
SPL {X  -160.798, Y  +338.700, Z    +0.000, E1   +25.294, E3 +257376.977}
SPL {X  -163.893, Y  +354.439, Z    +0.000, E1   +16.805, E3 +257371.451}
SPL {X  -165.158, Y  +365.746, Z    +0.000, E1   +10.198, E3 +257369.394}
SPL {X  -165.639, Y  +376.620, Z    +0.000, E1    +3.186, E3 +257369.194}
SPL {X  -165.650, Y  +380.533, Z    +0.000, E1    +0.120, E3 +257368.222}
SPL {X  -165.650, Y  +383.454, Z    +0.000, E1    -2.667, E3 +257367.629}
SPL {X  -165.650, Y  +388.792, Z    +0.000, E1    -9.482, E3 +257366.724}
SPL {X  -165.650, Y  +393.970, Z    +0.000, E1   -17.146, E3 +257365.880}
SPL {X  -165.650, Y  +401.614, Z    +0.000, E1   -27.619, E3 +257366.535}
SPL {X  -165.650, Y  +418.105, Z    +0.000, E1   -49.413, E3 +257361.943}
SPL {X  -165.650, Y  +465.736, Z    +0.000, E1   -65.678, E3 +257375.685}
SPL {X  -165.650, Y  +519.483, Z    +0.000, E1   -68.357, E3 +257401.870}
SPL {X  -165.650, Y  +548.869, Z    +0.000, E1   -62.199, E3 +257457.563}
ENDSPLINE

SPLINE
SPL {X  -165.650, Y  +534.780, Z    +0.000, E1   -57.803, E3 +257471.212}
ENDSPLINE

SPLINE
SPL {X  -165.650, Y  +545.905, Z    +0.000, E1   -57.853, E3 +257485.152}
SPL {X  -165.650, Y  +553.630, Z    +0.000, E1   -57.616, E3 +257496.601}
SPL {X  -165.650, Y  +563.473, Z    +0.000, E1   -57.690, E3 +257508.965}
SPL {X  -165.650, Y  +573.011, Z    +0.000, E1   -57.610, E3 +257521.757}
SPL {X  -165.650, Y  +581.530, Z    +0.000, E1   -57.678, E3 +257532.355}
SPL {X  -165.650, Y  +589.475, Z    +0.000, E1   -57.572, E3 +257543.341}
SPL {X  -165.650, Y  +599.695, Z    +0.000, E1   -57.964, E3 +257553.958}
SPL {X  -165.650, Y  +606.915, Z    +0.000, E1   -57.651, E3 +257565.314}
SPL {X  -165.650, Y  +614.927, Z    +0.000, E1   -57.517, E3 +257576.584}
SPL {X  -165.650, Y  +624.337, Z    +0.000, E1   -57.671, E3 +257587.810}
SPL {X  -165.650, Y  +634.236, Z    +0.000, E1   -57.671, E3 +257600.660}
SPL {X  -165.650, Y  +647.519, Z    +0.000, E1   -57.817, E3 +257616.988}
SPL {X  -165.650, Y  +657.986, Z    +0.000, E1   -57.646, E3 +257631.423}
SPL {X  -165.650, Y  +667.585, Z    +0.000, E1   -57.803, E3 +257642.819}
SPL {X  -165.634, Y  +677.794, Z    +0.000, E1   -57.650, E3 +257657.121}
SPL {X  -165.167, Y  +688.139, Z    +0.000, E1   -57.463, E3 +257671.701}
SPL {X  -164.009, Y  +698.761, Z    +0.000, E1   -57.613, E3 +257684.474}
SPL {X  -162.382, Y  +708.242, Z    +0.000, E1   -57.205, E3 +257699.400}
SPL {X  -160.577, Y  +716.182, Z    +0.000, E1   -56.676, E3 +257712.793}
SPL {X  -158.520, Y  +723.576, Z    +0.000, E1   -56.758, E3 +257721.838}
SPL {X  -156.858, Y  +728.749, Z    +0.000, E1   -56.333, E3 +257730.981}
SPL {X  -155.155, Y  +733.525, Z    +0.000, E1   -55.869, E3 +257739.757}
SPL {X  -153.442, Y  +737.914, Z    +0.000, E1   -55.562, E3 +257747.162}
SPL {X  -150.574, Y  +744.547, Z    +0.000, E1   -55.310, E3 +257757.145}
SPL {X  -147.713, Y  +750.471, Z    +0.000, E1   -54.514, E3 +257768.807}
SPL {X  -139.786, Y  +764.381, Z    +0.000, E1   -57.209, E3 +257772.995}
SPL {X  -110.324, Y  +799.066, Z    +0.000, E1   -54.396, E3 +257841.569}
SPL {X  -100.308, Y  +807.326, Z    +0.000, E1   -52.880, E3 +257886.137}
ENDSPLINE

SPLINE
SPL {X  -108.196, Y  +800.934, Z    +0.000, E1   -52.068, E3 +257978.463}
SPL {X  -144.673, Y  +756.182, Z    +0.000, E1   -41.752, E3 +257996.542}
SPL {X  -160.601, Y  +716.087, Z    +0.000, E1   -25.730, E3 +257996.170}
SPL {X  -164.850, Y  +691.761, Z    +0.000, E1   -12.424, E3 +257993.437}
SPL {X  -165.596, Y  +679.730, Z    +0.000, E1    -4.777, E3 +257992.311}
SPL {X  -165.650, Y  +674.376, Z    +0.000, E1    -0.866, E3 +257992.226}
SPL {X  -165.650, Y  +672.384, Z    +0.000, E1    +0.908, E3 +257991.107}
SPL {X  -165.650, Y  +669.093, Z    +0.000, E1    +4.549, E3 +257990.959}
SPL {X  -165.650, Y  +663.273, Z    +0.000, E1   +12.448, E3 +257990.196}
SPL {X  -165.650, Y  +654.885, Z    +0.000, E1   +25.204, E3 +257988.748}
SPL {X  -165.650, Y  +641.882, Z    +0.000, E1   +46.566, E3 +257981.619}
SPL {X  -165.650, Y  +630.946, Z    +0.000, E1   +55.779, E3 +257982.293}
SPL {X  -165.650, Y  +595.858, Z    +0.000, E1   +64.262, E3 +257997.174}
SPL {X  -165.650, Y  +589.368, Z    +0.000, E1   +58.232, E3 +258017.916}
SPL {X  -165.650, Y  +491.251, Z    +0.000, E1   +65.373, E3 +258074.342}
ENDSPLINE

SPLINE
SPL {X  -165.650, Y  +516.236, Z    +0.000, E1   +58.457, E3 +258095.023}
ENDSPLINE

SPLINE
SPL {X  -165.650, Y  +506.715, Z    +0.000, E1   +58.090, E3 +258109.476}
SPL {X  -165.650, Y  +496.085, Z    +0.000, E1   +57.984, E3 +258123.723}
SPL {X  -165.650, Y  +485.167, Z    +0.000, E1   +58.003, E3 +258137.555}
ENDSPLINE

SPLINE
SPL {X  -165.650, Y  +505.180, Z    +0.000, E1   +52.333, E3 +258144.307}
SPL {X  -165.650, Y  +506.534, Z    +0.000, E1   +50.148, E3 +258155.767}
ENDSPLINE

SPLINE
SPL {X  -165.650, Y  +495.166, Z    +0.000, E1   +51.070, E3 +258169.195}
SPL {X  -165.650, Y  +485.807, Z    +0.000, E1   +51.973, E3 +258178.928}
SPL {X  -165.650, Y  +475.672, Z    +0.000, E1   +52.573, E3 +258191.382}
SPL {X  -165.650, Y  +459.814, Z    +0.000, E1   +53.888, E3 +258207.571}
SPL {X  -165.650, Y  +448.876, Z    +0.000, E1   +54.452, E3 +258220.066}
SPL {X  -165.650, Y  +440.843, Z    +0.000, E1   +55.023, E3 +258228.130}
SPL {X  -165.650, Y  +431.771, Z    +0.000, E1   +55.549, E3 +258237.648}
SPL {X  -165.650, Y  +420.799, Z    +0.000, E1   +56.452, E3 +258247.034}
SPL {X  -165.650, Y  +409.731, Z    +0.000, E1   +57.273, E3 +258256.522}
SPL {X  -165.650, Y  +399.687, Z    +0.000, E1   +57.433, E3 +258268.706}
SPL {X  -165.650, Y  +388.492, Z    +0.000, E1   +57.709, E3 +258281.420}
SPL {X  -165.650, Y  +379.894, Z    +0.000, E1   +57.709, E3 +258292.523}
SPL {X  -165.538, Y  +372.423, Z    +0.000, E1   +57.528, E3 +258303.396}
SPL {X  -164.865, Y  +362.388, Z    +0.000, E1   +57.628, E3 +258315.783}
SPL {X  -163.867, Y  +354.258, Z    +0.000, E1   +57.359, E3 +258328.000}
SPL {X  -162.678, Y  +347.264, Z    +0.000, E1   +57.150, E3 +258338.341}
SPL {X  -161.618, Y  +342.173, Z    +0.000, E1   +56.783, E3 +258347.226}
SPL {X  -159.878, Y  +335.155, Z    +0.000, E1   +56.685, E3 +258357.030}
SPL {X  -158.009, Y  +328.771, Z    +0.000, E1   +56.325, E3 +258367.390}
SPL {X  -156.065, Y  +322.971, Z    +0.000, E1   +56.177, E3 +258375.734}
SPL {X  -154.487, Y  +318.719, Z    +0.000, E1   +55.733, E3 +258383.742}
SPL {X  -151.902, Y  +312.426, Z    +0.000, E1   +55.494, E3 +258393.217}
SPL {X  -148.935, Y  +305.985, Z    +0.000, E1   +54.737, E3 +258405.594}
SPL {X  -144.791, Y  +298.030, Z    +0.000, E1   +55.214, E3 +258413.327}
SPL {X  -133.590, Y  +280.553, Z    +0.000, E1   +59.642, E3 +258412.249}
SPL {X  -112.638, Y  +257.040, Z    +0.000, E1   +51.417, E3 +258515.633}
ENDSPLINE

SPLINE
SPL {X  -115.209, Y  +259.476, Z    +0.000, E1   +49.595, E3 +258548.903}
SPL {X  -147.344, Y  +302.806, Z    +0.000, E1   +40.158, E3 +258638.365}
SPL {X  -160.798, Y  +338.700, Z    +0.000, E1   +25.294, E3 +258637.847}
SPL {X  -163.893, Y  +354.439, Z    +0.000, E1   +16.805, E3 +258632.321}
SPL {X  -165.158, Y  +365.746, Z    +0.000, E1   +10.198, E3 +258630.264}
SPL {X  -165.580, Y  +373.688, Z    +0.000, E1    +5.094, E3 +258630.001}
SPL {X  -165.650, Y  +378.140, Z    +0.000, E1    +1.996, E3 +258630.087}
SPL {X  -165.650, Y  +381.477, Z    +0.000, E1    -0.622, E3 +258628.874}
SPL {X  -165.650, Y  +384.861, Z    +0.000, E1    -4.465, E3 +258628.277}
SPL {X  -165.650, Y  +388.792, Z    +0.000, E1    -9.482, E3 +258627.593}
SPL {X  -165.650, Y  +393.970, Z    +0.000, E1   -17.146, E3 +258626.750}
SPL {X  -165.650, Y  +401.614, Z    +0.000, E1   -27.619, E3 +258627.405}
SPL {X  -165.650, Y  +418.105, Z    +0.000, E1   -49.413, E3 +258622.813}
SPL {X  -165.650, Y  +465.736, Z    +0.000, E1   -65.678, E3 +258636.555}
SPL {X  -165.650, Y  +519.483, Z    +0.000, E1   -68.357, E3 +258662.740}
SPL {X  -165.650, Y  +548.869, Z    +0.000, E1   -62.199, E3 +258718.433}
ENDSPLINE

SPLINE
SPL {X  -165.650, Y  +534.780, Z    +0.000, E1   -57.803, E3 +258732.082}
ENDSPLINE

SPLINE
SPL {X  -165.650, Y  +545.905, Z    +0.000, E1   -57.853, E3 +258746.021}
SPL {X  -165.650, Y  +553.630, Z    +0.000, E1   -57.616, E3 +258757.471}
SPL {X  -165.650, Y  +563.473, Z    +0.000, E1   -57.690, E3 +258769.835}
SPL {X  -165.650, Y  +573.011, Z    +0.000, E1   -57.610, E3 +258782.626}
SPL {X  -165.650, Y  +581.530, Z    +0.000, E1   -57.678, E3 +258793.224}
SPL {X  -165.650, Y  +589.475, Z    +0.000, E1   -57.572, E3 +258804.211}
SPL {X  -165.650, Y  +599.695, Z    +0.000, E1   -57.964, E3 +258814.827}
SPL {X  -165.650, Y  +606.915, Z    +0.000, E1   -57.651, E3 +258826.184}
SPL {X  -165.650, Y  +614.927, Z    +0.000, E1   -57.517, E3 +258837.454}
SPL {X  -165.650, Y  +624.337, Z    +0.000, E1   -57.671, E3 +258848.680}
SPL {X  -165.650, Y  +634.236, Z    +0.000, E1   -57.671, E3 +258861.530}
SPL {X  -165.650, Y  +647.519, Z    +0.000, E1   -57.817, E3 +258877.857}
SPL {X  -165.650, Y  +657.986, Z    +0.000, E1   -57.646, E3 +258892.293}
SPL {X  -165.650, Y  +667.585, Z    +0.000, E1   -57.803, E3 +258903.689}
SPL {X  -165.634, Y  +677.794, Z    +0.000, E1   -57.650, E3 +258917.991}
SPL {X  -165.167, Y  +688.139, Z    +0.000, E1   -57.463, E3 +258932.570}
SPL {X  -164.009, Y  +698.761, Z    +0.000, E1   -57.613, E3 +258945.343}
SPL {X  -162.382, Y  +708.242, Z    +0.000, E1   -57.205, E3 +258960.269}
SPL {X  -160.577, Y  +716.182, Z    +0.000, E1   -56.676, E3 +258973.663}
SPL {X  -158.520, Y  +723.576, Z    +0.000, E1   -56.758, E3 +258982.708}
SPL {X  -156.858, Y  +728.749, Z    +0.000, E1   -56.333, E3 +258991.850}
SPL {X  -155.155, Y  +733.525, Z    +0.000, E1   -55.869, E3 +259000.627}
SPL {X  -152.530, Y  +740.111, Z    +0.000, E1   -55.545, E3 +259011.103}
SPL {X  -149.838, Y  +746.130, Z    +0.000, E1   -55.135, E3 +259020.823}
SPL {X  -147.713, Y  +750.471, Z    +0.000, E1   -54.514, E3 +259029.677}
SPL {X  -139.786, Y  +764.381, Z    +0.000, E1   -57.209, E3 +259033.865}
SPL {X  -110.324, Y  +799.066, Z    +0.000, E1   -54.396, E3 +259102.439}
SPL {X  -100.308, Y  +807.326, Z    +0.000, E1   -52.880, E3 +259147.006}
ENDSPLINE

SPLINE
SPL {X  -108.196, Y  +800.934, Z    +0.000, E1   -52.068, E3 +259239.333}
SPL {X  -144.673, Y  +756.182, Z    +0.000, E1   -41.752, E3 +259257.412}
SPL {X  -160.601, Y  +716.087, Z    +0.000, E1   -25.730, E3 +259257.039}
SPL {X  -164.850, Y  +691.761, Z    +0.000, E1   -12.424, E3 +259254.307}
SPL {X  -165.596, Y  +679.730, Z    +0.000, E1    -4.777, E3 +259253.180}
SPL {X  -165.650, Y  +674.376, Z    +0.000, E1    -0.866, E3 +259253.096}
SPL {X  -165.650, Y  +672.384, Z    +0.000, E1    +0.908, E3 +259251.977}
SPL {X  -165.650, Y  +669.968, Z    +0.000, E1    +3.584, E3 +259251.793}
SPL {X  -165.650, Y  +666.667, Z    +0.000, E1    +7.761, E3 +259251.472}
SPL {X  -165.650, Y  +662.028, Z    +0.000, E1   +14.359, E3 +259251.102}
SPL {X  -165.650, Y  +654.885, Z    +0.000, E1   +25.204, E3 +259249.617}
SPL {X  -165.650, Y  +641.882, Z    +0.000, E1   +46.566, E3 +259242.488}
SPL {X  -165.650, Y  +630.946, Z    +0.000, E1   +55.779, E3 +259243.163}
SPL {X  -165.650, Y  +590.135, Z    +0.000, E1   +59.110, E3 +259275.783}
SPL {X  -165.650, Y  +491.251, Z    +0.000, E1   +65.373, E3 +259335.212}
ENDSPLINE

SPLINE
SPL {X  -165.650, Y  +516.236, Z    +0.000, E1   +58.457, E3 +259355.892}
ENDSPLINE

SPLINE
SPL {X  -165.650, Y  +506.715, Z    +0.000, E1   +58.090, E3 +259370.345}
SPL {X  -165.650, Y  +496.085, Z    +0.000, E1   +57.984, E3 +259384.593}
SPL {X  -165.650, Y  +485.167, Z    +0.000, E1   +58.003, E3 +259398.425}
ENDSPLINE

SPLINE
SPL {X  -165.650, Y  +505.180, Z    +0.000, E1   +52.333, E3 +259405.177}
SPL {X  -165.650, Y  +506.534, Z    +0.000, E1   +50.148, E3 +259416.636}
ENDSPLINE

SPLINE
SPL {X  -165.650, Y  +495.166, Z    +0.000, E1   +51.070, E3 +259430.065}
SPL {X  -165.650, Y  +485.807, Z    +0.000, E1   +51.973, E3 +259439.798}
SPL {X  -165.650, Y  +478.030, Z    +0.000, E1   +52.389, E3 +259449.604}
SPL {X  -165.650, Y  +467.527, Z    +0.000, E1   +53.334, E3 +259460.099}
SPL {X  -165.650, Y  +457.379, Z    +0.000, E1   +53.935, E3 +259471.642}
SPL {X  -165.650, Y  +444.120, Z    +0.000, E1   +54.815, E3 +259485.688}
SPL {X  -165.650, Y  +431.771, Z    +0.000, E1   +55.549, E3 +259498.518}
SPL {X  -165.650, Y  +420.799, Z    +0.000, E1   +56.452, E3 +259507.903}
SPL {X  -165.650, Y  +409.731, Z    +0.000, E1   +57.273, E3 +259517.392}
SPL {X  -165.650, Y  +399.687, Z    +0.000, E1   +57.433, E3 +259529.576}
SPL {X  -165.650, Y  +388.492, Z    +0.000, E1   +57.709, E3 +259542.289}
SPL {X  -165.650, Y  +379.894, Z    +0.000, E1   +57.709, E3 +259553.393}
SPL {X  -165.538, Y  +372.423, Z    +0.000, E1   +57.528, E3 +259564.266}
SPL {X  -164.865, Y  +362.388, Z    +0.000, E1   +57.628, E3 +259576.652}
SPL {X  -163.867, Y  +354.258, Z    +0.000, E1   +57.359, E3 +259588.869}
SPL {X  -162.678, Y  +347.264, Z    +0.000, E1   +57.150, E3 +259599.211}
SPL {X  -161.618, Y  +342.173, Z    +0.000, E1   +56.783, E3 +259608.096}
SPL {X  -159.878, Y  +335.155, Z    +0.000, E1   +56.685, E3 +259617.900}
SPL {X  -158.009, Y  +328.771, Z    +0.000, E1   +56.325, E3 +259628.259}
SPL {X  -156.065, Y  +322.971, Z    +0.000, E1   +56.177, E3 +259636.603}
SPL {X  -154.487, Y  +318.719, Z    +0.000, E1   +55.733, E3 +259644.612}
SPL {X  -151.902, Y  +312.426, Z    +0.000, E1   +55.494, E3 +259654.087}
SPL {X  -149.742, Y  +307.668, Z    +0.000, E1   +54.896, E3 +259663.299}
SPL {X  -146.487, Y  +301.160, Z    +0.000, E1   +54.808, E3 +259672.162}
SPL {X  -133.590, Y  +280.553, Z    +0.000, E1   +59.642, E3 +259673.119}
SPL {X  -112.638, Y  +257.040, Z    +0.000, E1   +51.417, E3 +259776.502}
ENDSPLINE

SPLINE
SPL {X  -115.209, Y  +259.476, Z    +0.000, E1   +49.595, E3 +259809.772}
SPL {X  -147.344, Y  +302.806, Z    +0.000, E1   +40.158, E3 +259899.235}
SPL {X  -160.798, Y  +338.700, Z    +0.000, E1   +25.294, E3 +259898.717}
SPL {X  -163.893, Y  +354.439, Z    +0.000, E1   +16.805, E3 +259893.191}
SPL {X  -165.158, Y  +365.746, Z    +0.000, E1   +10.198, E3 +259891.133}
SPL {X  -165.639, Y  +376.620, Z    +0.000, E1    +3.186, E3 +259890.933}
SPL {X  -165.650, Y  +381.477, Z    +0.000, E1    -0.622, E3 +259889.744}
SPL {X  -165.650, Y  +386.363, Z    +0.000, E1    -6.162, E3 +259889.093}
SPL {X  -165.650, Y  +392.511, Z    +0.000, E1   -14.940, E3 +259887.533}
SPL {X  -165.650, Y  +398.939, Z    +0.000, E1   -23.851, E3 +259888.918}
SPL {X  -165.650, Y  +404.249, Z    +0.000, E1   -31.650, E3 +259887.639}
SPL {X  -165.650, Y  +418.105, Z    +0.000, E1   -49.413, E3 +259883.682}
SPL {X  -165.650, Y  +465.736, Z    +0.000, E1   -65.678, E3 +259897.425}
SPL {X  -165.650, Y  +519.483, Z    +0.000, E1   -68.357, E3 +259923.609}
SPL {X  -165.650, Y  +548.869, Z    +0.000, E1   -62.199, E3 +259979.302}
ENDSPLINE

SPLINE
SPL {X  -165.650, Y  +530.735, Z    +0.000, E1   -57.778, E3 +259987.726}
ENDSPLINE

SPLINE
SPL {X  -165.650, Y  +536.777, Z    +0.000, E1   -57.774, E3 +259995.603}
SPL {X  -165.650, Y  +545.905, Z    +0.000, E1   -57.853, E3 +260006.891}
SPL {X  -165.650, Y  +553.630, Z    +0.000, E1   -57.616, E3 +260018.340}
SPL {X  -165.650, Y  +563.473, Z    +0.000, E1   -57.690, E3 +260030.705}
SPL {X  -165.650, Y  +573.011, Z    +0.000, E1   -57.610, E3 +260043.496}
SPL {X  -165.650, Y  +581.530, Z    +0.000, E1   -57.678, E3 +260054.094}
SPL {X  -165.650, Y  +589.475, Z    +0.000, E1   -57.572, E3 +260065.081}
SPL {X  -165.650, Y  +599.695, Z    +0.000, E1   -57.964, E3 +260075.697}
SPL {X  -165.650, Y  +606.915, Z    +0.000, E1   -57.651, E3 +260087.053}
SPL {X  -165.650, Y  +614.927, Z    +0.000, E1   -57.517, E3 +260098.323}
SPL {X  -165.650, Y  +624.337, Z    +0.000, E1   -57.671, E3 +260109.549}
SPL {X  -165.650, Y  +634.236, Z    +0.000, E1   -57.671, E3 +260122.399}
SPL {X  -165.650, Y  +647.519, Z    +0.000, E1   -57.817, E3 +260138.727}
SPL {X  -165.650, Y  +657.986, Z    +0.000, E1   -57.646, E3 +260153.162}
SPL {X  -165.650, Y  +667.585, Z    +0.000, E1   -57.803, E3 +260164.558}
SPL {X  -165.634, Y  +677.794, Z    +0.000, E1   -57.650, E3 +260178.860}
SPL {X  -165.167, Y  +688.139, Z    +0.000, E1   -57.463, E3 +260193.440}
SPL {X  -164.323, Y  +696.426, Z    +0.000, E1   -57.565, E3 +260203.427}
SPL {X  -163.313, Y  +703.224, Z    +0.000, E1   -57.403, E3 +260213.320}
SPL {X  -161.906, Y  +710.520, Z    +0.000, E1   -57.149, E3 +260224.272}
SPL {X  -160.577, Y  +716.182, Z    +0.000, E1   -56.676, E3 +260234.533}
SPL {X  -158.520, Y  +723.576, Z    +0.000, E1   -56.758, E3 +260243.577}
SPL {X  -156.858, Y  +728.749, Z    +0.000, E1   -56.333, E3 +260252.720}
SPL {X  -155.155, Y  +733.525, Z    +0.000, E1   -55.869, E3 +260261.496}
SPL {X  -153.442, Y  +737.914, Z    +0.000, E1   -55.562, E3 +260268.901}
SPL {X  -150.574, Y  +744.547, Z    +0.000, E1   -55.310, E3 +260278.884}
SPL {X  -147.713, Y  +750.471, Z    +0.000, E1   -54.514, E3 +260290.546}
SPL {X  -139.786, Y  +764.381, Z    +0.000, E1   -57.209, E3 +260294.734}
SPL {X  -110.324, Y  +799.066, Z    +0.000, E1   -54.396, E3 +260363.309}
SPL {X  -100.308, Y  +807.326, Z    +0.000, E1   -52.880, E3 +260407.876}
ENDSPLINE

SPLINE
SPL {X  -108.196, Y  +800.934, Z    +0.000, E1   -52.068, E3 +260500.202}
SPL {X  -144.673, Y  +756.182, Z    +0.000, E1   -41.752, E3 +260518.281}
SPL {X  -160.601, Y  +716.087, Z    +0.000, E1   -25.730, E3 +260517.909}
SPL {X  -164.850, Y  +691.761, Z    +0.000, E1   -12.424, E3 +260515.176}
SPL {X  -165.596, Y  +679.730, Z    +0.000, E1    -4.777, E3 +260514.050}
SPL {X  -165.650, Y  +674.376, Z    +0.000, E1    -0.866, E3 +260513.965}
SPL {X  -165.650, Y  +672.384, Z    +0.000, E1    +0.908, E3 +260512.846}
SPL {X  -165.650, Y  +669.093, Z    +0.000, E1    +4.549, E3 +260512.698}
SPL {X  -165.650, Y  +663.273, Z    +0.000, E1   +12.448, E3 +260511.935}
SPL {X  -165.650, Y  +654.885, Z    +0.000, E1   +25.204, E3 +260510.487}
SPL {X  -165.650, Y  +641.882, Z    +0.000, E1   +46.566, E3 +260503.358}
SPL {X  -165.650, Y  +630.946, Z    +0.000, E1   +55.779, E3 +260504.032}
SPL {X  -165.650, Y  +590.135, Z    +0.000, E1   +59.110, E3 +260536.652}
SPL {X  -165.650, Y  +491.251, Z    +0.000, E1   +65.373, E3 +260596.081}
ENDSPLINE

SPLINE
SPL {X  -165.650, Y  +517.534, Z    +0.000, E1   +59.090, E3 +260610.679}
ENDSPLINE

SPLINE
SPL {X  -165.650, Y  +515.821, Z    +0.000, E1   +58.153, E3 +260619.126}
SPL {X  -165.650, Y  +506.715, Z    +0.000, E1   +58.090, E3 +260631.215}
SPL {X  -165.650, Y  +496.085, Z    +0.000, E1   +57.984, E3 +260645.462}
SPL {X  -165.650, Y  +485.167, Z    +0.000, E1   +58.003, E3 +260659.294}
ENDSPLINE

SPLINE
SPL {X  -165.650, Y  +505.180, Z    +0.000, E1   +52.333, E3 +260666.046}
SPL {X  -165.650, Y  +506.534, Z    +0.000, E1   +50.148, E3 +260677.506}
ENDSPLINE

SPLINE
SPL {X  -165.650, Y  +495.166, Z    +0.000, E1   +51.070, E3 +260690.934}
SPL {X  -165.650, Y  +485.807, Z    +0.000, E1   +51.973, E3 +260700.667}
SPL {X  -165.650, Y  +478.030, Z    +0.000, E1   +52.389, E3 +260710.474}
SPL {X  -165.650, Y  +467.527, Z    +0.000, E1   +53.334, E3 +260720.968}
SPL {X  -165.650, Y  +453.744, Z    +0.000, E1   +54.190, E3 +260736.449}
SPL {X  -165.650, Y  +440.843, Z    +0.000, E1   +55.023, E3 +260749.869}
SPL {X  -165.650, Y  +431.771, Z    +0.000, E1   +55.549, E3 +260759.387}
SPL {X  -165.650, Y  +420.799, Z    +0.000, E1   +56.452, E3 +260768.773}
SPL {X  -165.650, Y  +409.731, Z    +0.000, E1   +57.273, E3 +260778.261}
SPL {X  -165.650, Y  +399.687, Z    +0.000, E1   +57.433, E3 +260790.446}
SPL {X  -165.650, Y  +388.492, Z    +0.000, E1   +57.709, E3 +260803.159}
SPL {X  -165.650, Y  +379.894, Z    +0.000, E1   +57.709, E3 +260814.263}
SPL {X  -165.399, Y  +369.388, Z    +0.000, E1   +57.657, E3 +260828.356}
SPL {X  -164.717, Y  +360.945, Z    +0.000, E1   +57.468, E3 +260840.294}
SPL {X  -163.867, Y  +354.258, Z    +0.000, E1   +57.359, E3 +260849.739}
SPL {X  -162.678, Y  +347.264, Z    +0.000, E1   +57.150, E3 +260860.080}
SPL {X  -161.618, Y  +342.173, Z    +0.000, E1   +56.783, E3 +260868.966}
SPL {X  -159.878, Y  +335.155, Z    +0.000, E1   +56.685, E3 +260878.769}
SPL {X  -158.009, Y  +328.771, Z    +0.000, E1   +56.325, E3 +260889.129}
SPL {X  -156.065, Y  +322.971, Z    +0.000, E1   +56.177, E3 +260897.473}
SPL {X  -153.731, Y  +316.803, Z    +0.000, E1   +55.737, E3 +260908.049}
SPL {X  -150.320, Y  +308.902, Z    +0.000, E1   +55.085, E3 +260921.745}
SPL {X  -147.957, Y  +304.011, Z    +0.000, E1   +54.431, E3 +260931.208}
SPL {X  -144.791, Y  +298.030, Z    +0.000, E1   +55.214, E3 +260935.066}
SPL {X  -133.590, Y  +280.553, Z    +0.000, E1   +59.642, E3 +260933.988}
SPL {X  -112.638, Y  +257.040, Z    +0.000, E1   +51.417, E3 +261037.372}
ENDSPLINE

SPLINE
SPL {X  -115.209, Y  +259.476, Z    +0.000, E1   +49.595, E3 +261070.642}
SPL {X  -147.344, Y  +302.806, Z    +0.000, E1   +40.158, E3 +261160.104}
SPL {X  -160.798, Y  +338.700, Z    +0.000, E1   +25.294, E3 +261159.586}
SPL {X  -163.893, Y  +354.439, Z    +0.000, E1   +16.805, E3 +261154.060}
SPL {X  -165.158, Y  +365.746, Z    +0.000, E1   +10.198, E3 +261152.003}
SPL {X  -165.580, Y  +373.688, Z    +0.000, E1    +5.094, E3 +261151.740}
SPL {X  -165.650, Y  +379.719, Z    +0.000, E1    +0.894, E3 +261151.170}
SPL {X  -165.650, Y  +383.454, Z    +0.000, E1    -2.667, E3 +261150.238}
SPL {X  -165.650, Y  +387.779, Z    +0.000, E1    -8.159, E3 +261149.911}
SPL {X  -165.650, Y  +392.511, Z    +0.000, E1   -14.940, E3 +261148.402}
SPL {X  -165.650, Y  +401.614, Z    +0.000, E1   -27.619, E3 +261149.144}
SPL {X  -165.650, Y  +418.105, Z    +0.000, E1   -49.413, E3 +261144.552}
SPL {X  -165.650, Y  +465.736, Z    +0.000, E1   -65.678, E3 +261158.294}
SPL {X  -165.650, Y  +519.483, Z    +0.000, E1   -68.357, E3 +261184.479}
SPL {X  -165.650, Y  +548.869, Z    +0.000, E1   -62.199, E3 +261240.172}
ENDSPLINE

SPLINE
SPL {X  -165.650, Y  +534.780, Z    +0.000, E1   -57.803, E3 +261253.821}
ENDSPLINE

SPLINE
SPL {X  -165.650, Y  +545.905, Z    +0.000, E1   -57.853, E3 +261267.760}
SPL {X  -165.650, Y  +555.746, Z    +0.000, E1   -57.571, E3 +261282.398}
SPL {X  -165.650, Y  +566.557, Z    +0.000, E1   -57.834, E3 +261294.526}
SPL {X  -165.650, Y  +573.011, Z    +0.000, E1   -57.610, E3 +261304.365}
SPL {X  -165.650, Y  +581.530, Z    +0.000, E1   -57.678, E3 +261314.963}
SPL {X  -165.650, Y  +589.475, Z    +0.000, E1   -57.572, E3 +261325.950}
SPL {X  -165.650, Y  +599.695, Z    +0.000, E1   -57.964, E3 +261336.566}
SPL {X  -165.650, Y  +606.915, Z    +0.000, E1   -57.651, E3 +261347.923}
SPL {X  -165.650, Y  +614.927, Z    +0.000, E1   -57.517, E3 +261359.193}
SPL {X  -165.650, Y  +624.337, Z    +0.000, E1   -57.671, E3 +261370.419}
SPL {X  -165.650, Y  +634.236, Z    +0.000, E1   -57.671, E3 +261383.269}
SPL {X  -165.650, Y  +647.519, Z    +0.000, E1   -57.817, E3 +261399.596}
SPL {X  -165.650, Y  +657.986, Z    +0.000, E1   -57.646, E3 +261414.032}
SPL {X  -165.650, Y  +667.585, Z    +0.000, E1   -57.803, E3 +261425.428}
SPL {X  -165.634, Y  +677.794, Z    +0.000, E1   -57.650, E3 +261439.730}
SPL {X  -165.167, Y  +688.139, Z    +0.000, E1   -57.463, E3 +261454.309}
SPL {X  -164.009, Y  +698.761, Z    +0.000, E1   -57.613, E3 +261467.082}
SPL {X  -162.382, Y  +708.242, Z    +0.000, E1   -57.205, E3 +261482.008}
SPL {X  -160.577, Y  +716.182, Z    +0.000, E1   -56.676, E3 +261495.402}
SPL {X  -158.520, Y  +723.576, Z    +0.000, E1   -56.758, E3 +261504.447}
SPL {X  -156.858, Y  +728.749, Z    +0.000, E1   -56.333, E3 +261513.589}
SPL {X  -155.155, Y  +733.525, Z    +0.000, E1   -55.869, E3 +261522.366}
SPL {X  -152.530, Y  +740.111, Z    +0.000, E1   -55.545, E3 +261532.842}
SPL {X  -149.838, Y  +746.130, Z    +0.000, E1   -55.135, E3 +261542.563}
SPL {X  -147.713, Y  +750.471, Z    +0.000, E1   -54.514, E3 +261551.416}
SPL {X  -139.786, Y  +764.381, Z    +0.000, E1   -57.209, E3 +261555.604}
SPL {X  -110.324, Y  +799.066, Z    +0.000, E1   -54.396, E3 +261624.178}
SPL {X  -100.308, Y  +807.326, Z    +0.000, E1   -52.880, E3 +261668.745}
ENDSPLINE

SPLINE
SPL {X  -108.196, Y  +800.934, Z    +0.000, E1   -52.068, E3 +261761.072}
SPL {X  -147.753, Y  +750.393, Z    +0.000, E1   -39.863, E3 +261779.294}
SPL {X  -161.414, Y  +712.720, Z    +0.000, E1   -24.024, E3 +261778.636}
SPL {X  -164.278, Y  +696.774, Z    +0.000, E1   -15.225, E3 +261773.248}
SPL {X  -165.078, Y  +689.251, Z    +0.000, E1   -10.876, E3 +261777.400}
SPL {X  -165.596, Y  +679.730, Z    +0.000, E1    -4.777, E3 +261774.919}
SPL {X  -165.650, Y  +674.376, Z    +0.000, E1    -0.866, E3 +261774.835}
SPL {X  -165.650, Y  +672.384, Z    +0.000, E1    +0.908, E3 +261773.716}
SPL {X  -165.650, Y  +669.093, Z    +0.000, E1    +4.549, E3 +261773.567}
SPL {X  -165.650, Y  +663.273, Z    +0.000, E1   +12.448, E3 +261772.804}
SPL {X  -165.650, Y  +657.199, Z    +0.000, E1   +21.720, E3 +261772.074}
SPL {X  -165.650, Y  +652.963, Z    +0.000, E1   +28.395, E3 +261770.759}
SPL {X  -165.650, Y  +641.882, Z    +0.000, E1   +46.566, E3 +261764.227}
SPL {X  -165.650, Y  +630.946, Z    +0.000, E1   +55.779, E3 +261764.902}
SPL {X  -165.650, Y  +590.135, Z    +0.000, E1   +59.110, E3 +261797.522}
SPL {X  -165.650, Y  +491.251, Z    +0.000, E1   +65.373, E3 +261856.951}
ENDSPLINE

SPLINE
SPL {X  -165.650, Y  +516.236, Z    +0.000, E1   +58.457, E3 +261877.632}
ENDSPLINE

SPLINE
SPL {X  -165.650, Y  +506.715, Z    +0.000, E1   +58.090, E3 +261892.085}
SPL {X  -165.650, Y  +496.085, Z    +0.000, E1   +57.984, E3 +261906.332}
SPL {X  -165.650, Y  +485.167, Z    +0.000, E1   +58.003, E3 +261920.164}
ENDSPLINE

SPLINE
SPL {X  -165.650, Y  +505.180, Z    +0.000, E1   +52.333, E3 +261926.916}
SPL {X  -165.650, Y  +506.534, Z    +0.000, E1   +50.148, E3 +261938.375}
ENDSPLINE

SPLINE
SPL {X  -165.650, Y  +495.166, Z    +0.000, E1   +51.070, E3 +261951.804}
SPL {X  -165.650, Y  +485.807, Z    +0.000, E1   +51.973, E3 +261961.537}
SPL {X  -165.650, Y  +475.672, Z    +0.000, E1   +52.573, E3 +261973.990}
SPL {X  -165.650, Y  +459.814, Z    +0.000, E1   +53.888, E3 +261990.180}
SPL {X  -165.650, Y  +448.876, Z    +0.000, E1   +54.452, E3 +262002.674}
SPL {X  -165.650, Y  +440.843, Z    +0.000, E1   +55.023, E3 +262010.739}
SPL {X  -165.650, Y  +431.771, Z    +0.000, E1   +55.549, E3 +262020.257}
SPL {X  -165.650, Y  +420.799, Z    +0.000, E1   +56.452, E3 +262029.642}
SPL {X  -165.650, Y  +406.746, Z    +0.000, E1   +57.489, E3 +262041.687}
SPL {X  -165.650, Y  +399.455, Z    +0.000, E1   +57.184, E3 +262053.109}
SPL {X  -165.650, Y  +388.492, Z    +0.000, E1   +57.709, E3 +262064.028}
SPL {X  -165.650, Y  +379.894, Z    +0.000, E1   +57.709, E3 +262075.132}
SPL {X  -165.399, Y  +369.388, Z    +0.000, E1   +57.657, E3 +262089.226}
SPL {X  -164.717, Y  +360.945, Z    +0.000, E1   +57.468, E3 +262101.164}
SPL {X  -163.867, Y  +354.258, Z    +0.000, E1   +57.359, E3 +262110.608}
SPL {X  -162.678, Y  +347.264, Z    +0.000, E1   +57.150, E3 +262120.950}
SPL {X  -160.825, Y  +338.812, Z    +0.000, E1   +56.892, E3 +262133.692}
SPL {X  -158.481, Y  +330.294, Z    +0.000, E1   +56.303, E3 +262148.210}
SPL {X  -156.065, Y  +322.971, Z    +0.000, E1   +56.177, E3 +262158.342}
SPL {X  -154.487, Y  +318.719, Z    +0.000, E1   +55.733, E3 +262166.351}
SPL {X  -151.902, Y  +312.426, Z    +0.000, E1   +55.494, E3 +262175.826}
SPL {X  -148.935, Y  +305.985, Z    +0.000, E1   +54.737, E3 +262188.203}
SPL {X  -144.791, Y  +298.030, Z    +0.000, E1   +55.214, E3 +262195.935}
SPL {X  -133.590, Y  +280.553, Z    +0.000, E1   +59.642, E3 +262194.858}
SPL {X  -112.638, Y  +257.040, Z    +0.000, E1   +51.417, E3 +262298.241}
ENDSPLINE

SPLINE
SPL {X  -115.209, Y  +259.476, Z    +0.000, E1   +49.595, E3 +262331.512}
SPL {X  -147.344, Y  +302.806, Z    +0.000, E1   +40.158, E3 +262420.974}
SPL {X  -160.798, Y  +338.700, Z    +0.000, E1   +25.294, E3 +262420.456}
SPL {X  -163.893, Y  +354.439, Z    +0.000, E1   +16.805, E3 +262414.930}
SPL {X  -165.158, Y  +365.746, Z    +0.000, E1   +10.198, E3 +262412.872}
SPL {X  -165.639, Y  +376.620, Z    +0.000, E1    +3.186, E3 +262412.673}
SPL {X  -165.650, Y  +380.533, Z    +0.000, E1    +0.120, E3 +262411.701}
SPL {X  -165.650, Y  +383.454, Z    +0.000, E1    -2.667, E3 +262411.108}
SPL {X  -165.650, Y  +388.792, Z    +0.000, E1    -9.482, E3 +262410.202}
SPL {X  -165.650, Y  +393.970, Z    +0.000, E1   -17.146, E3 +262409.358}
SPL {X  -165.650, Y  +401.614, Z    +0.000, E1   -27.619, E3 +262410.013}
SPL {X  -165.650, Y  +418.105, Z    +0.000, E1   -49.413, E3 +262405.421}
SPL {X  -165.650, Y  +465.736, Z    +0.000, E1   -65.678, E3 +262419.164}
SPL {X  -165.650, Y  +519.483, Z    +0.000, E1   -68.357, E3 +262445.349}
SPL {X  -165.650, Y  +548.869, Z    +0.000, E1   -62.199, E3 +262501.041}
ENDSPLINE

SPLINE
SPL {X  -165.650, Y  +534.780, Z    +0.000, E1   -57.803, E3 +262514.691}
ENDSPLINE

SPLINE
SPL {X  -165.650, Y  +545.905, Z    +0.000, E1   -57.853, E3 +262528.630}
SPL {X  -165.650, Y  +553.630, Z    +0.000, E1   -57.616, E3 +262540.079}
SPL {X  -165.650, Y  +563.473, Z    +0.000, E1   -57.690, E3 +262552.444}
SPL {X  -165.650, Y  +573.011, Z    +0.000, E1   -57.610, E3 +262565.235}
SPL {X  -165.650, Y  +581.530, Z    +0.000, E1   -57.678, E3 +262575.833}
SPL {X  -165.650, Y  +589.475, Z    +0.000, E1   -57.572, E3 +262586.820}
SPL {X  -165.650, Y  +599.695, Z    +0.000, E1   -57.964, E3 +262597.436}
SPL {X  -165.650, Y  +606.915, Z    +0.000, E1   -57.651, E3 +262608.793}
SPL {X  -165.650, Y  +614.927, Z    +0.000, E1   -57.517, E3 +262620.062}
SPL {X  -165.650, Y  +624.337, Z    +0.000, E1   -57.671, E3 +262631.288}
SPL {X  -165.650, Y  +634.236, Z    +0.000, E1   -57.671, E3 +262644.139}
SPL {X  -165.650, Y  +647.519, Z    +0.000, E1   -57.817, E3 +262660.466}
SPL {X  -165.650, Y  +657.986, Z    +0.000, E1   -57.646, E3 +262674.901}
SPL {X  -165.650, Y  +667.585, Z    +0.000, E1   -57.803, E3 +262686.297}
SPL {X  -165.634, Y  +677.794, Z    +0.000, E1   -57.650, E3 +262700.599}
SPL {X  -165.167, Y  +688.139, Z    +0.000, E1   -57.463, E3 +262715.179}
SPL {X  -164.009, Y  +698.761, Z    +0.000, E1   -57.613, E3 +262727.952}
SPL {X  -162.382, Y  +708.242, Z    +0.000, E1   -57.205, E3 +262742.878}
SPL {X  -160.577, Y  +716.182, Z    +0.000, E1   -56.676, E3 +262756.272}
SPL {X  -158.520, Y  +723.576, Z    +0.000, E1   -56.758, E3 +262765.316}
SPL {X  -156.858, Y  +728.749, Z    +0.000, E1   -56.333, E3 +262774.459}
SPL {X  -155.155, Y  +733.525, Z    +0.000, E1   -55.869, E3 +262783.236}
SPL {X  -153.442, Y  +737.914, Z    +0.000, E1   -55.562, E3 +262790.640}
SPL {X  -150.574, Y  +744.547, Z    +0.000, E1   -55.310, E3 +262800.623}
SPL {X  -147.713, Y  +750.471, Z    +0.000, E1   -54.514, E3 +262812.285}
SPL {X  -139.786, Y  +764.381, Z    +0.000, E1   -57.209, E3 +262816.474}
SPL {X  -110.324, Y  +799.066, Z    +0.000, E1   -54.396, E3 +262885.048}
SPL {X  -100.308, Y  +807.326, Z    +0.000, E1   -52.880, E3 +262929.615}
ENDSPLINE

SPLINE
SPL {X  -108.196, Y  +800.934, Z    +0.000, E1   -52.068, E3 +263021.941}
SPL {X  -144.673, Y  +756.182, Z    +0.000, E1   -41.752, E3 +263040.020}
SPL {X  -160.601, Y  +716.087, Z    +0.000, E1   -25.730, E3 +263039.648}
SPL {X  -164.850, Y  +691.761, Z    +0.000, E1   -12.424, E3 +263036.915}
SPL {X  -165.596, Y  +679.730, Z    +0.000, E1    -4.777, E3 +263035.789}
SPL {X  -165.650, Y  +674.376, Z    +0.000, E1    -0.866, E3 +263035.704}
SPL {X  -165.650, Y  +672.384, Z    +0.000, E1    +0.908, E3 +263034.585}
SPL {X  -165.650, Y  +669.093, Z    +0.000, E1    +4.549, E3 +263034.437}
SPL {X  -165.650, Y  +663.273, Z    +0.000, E1   +12.448, E3 +263033.674}
SPL {X  -165.650, Y  +654.885, Z    +0.000, E1   +25.204, E3 +263032.226}
SPL {X  -165.650, Y  +641.882, Z    +0.000, E1   +46.566, E3 +263025.097}
SPL {X  -165.650, Y  +630.946, Z    +0.000, E1   +55.779, E3 +263025.772}
SPL {X  -165.650, Y  +595.858, Z    +0.000, E1   +64.262, E3 +263040.652}
SPL {X  -165.650, Y  +589.368, Z    +0.000, E1   +58.232, E3 +263061.394}
SPL {X  -165.650, Y  +491.251, Z    +0.000, E1   +65.373, E3 +263117.821}
ENDSPLINE

SPLINE
SPL {X  -165.650, Y  +516.236, Z    +0.000, E1   +58.457, E3 +263138.501}
ENDSPLINE

SPLINE
SPL {X  -165.650, Y  +506.715, Z    +0.000, E1   +58.090, E3 +263152.954}
SPL {X  -165.650, Y  +496.085, Z    +0.000, E1   +57.984, E3 +263167.201}
SPL {X  -165.650, Y  +485.167, Z    +0.000, E1   +58.003, E3 +263181.033}
ENDSPLINE

SPLINE
SPL {X  -165.650, Y  +505.180, Z    +0.000, E1   +52.333, E3 +263187.785}
SPL {X  -165.650, Y  +506.534, Z    +0.000, E1   +50.148, E3 +263199.245}
ENDSPLINE

SPLINE
SPL {X  -165.650, Y  +495.166, Z    +0.000, E1   +51.070, E3 +263212.673}
SPL {X  -165.650, Y  +485.807, Z    +0.000, E1   +51.973, E3 +263222.406}
SPL {X  -165.650, Y  +475.672, Z    +0.000, E1   +52.573, E3 +263234.860}
SPL {X  -165.650, Y  +459.814, Z    +0.000, E1   +53.888, E3 +263251.049}
SPL {X  -165.650, Y  +448.876, Z    +0.000, E1   +54.452, E3 +263263.544}
SPL {X  -165.650, Y  +440.843, Z    +0.000, E1   +55.023, E3 +263271.608}
SPL {X  -165.650, Y  +431.771, Z    +0.000, E1   +55.549, E3 +263281.126}
SPL {X  -165.650, Y  +420.799, Z    +0.000, E1   +56.452, E3 +263290.512}
SPL {X  -165.650, Y  +409.731, Z    +0.000, E1   +57.273, E3 +263300.000}
SPL {X  -165.650, Y  +399.687, Z    +0.000, E1   +57.433, E3 +263312.185}
SPL {X  -165.650, Y  +388.492, Z    +0.000, E1   +57.709, E3 +263324.898}
SPL {X  -165.650, Y  +379.894, Z    +0.000, E1   +57.709, E3 +263336.002}
SPL {X  -165.538, Y  +372.423, Z    +0.000, E1   +57.528, E3 +263346.875}
SPL {X  -164.865, Y  +362.388, Z    +0.000, E1   +57.628, E3 +263359.261}
SPL {X  -163.867, Y  +354.258, Z    +0.000, E1   +57.359, E3 +263371.478}
SPL {X  -162.678, Y  +347.264, Z    +0.000, E1   +57.150, E3 +263381.819}
SPL {X  -161.618, Y  +342.173, Z    +0.000, E1   +56.783, E3 +263390.705}
SPL {X  -159.878, Y  +335.155, Z    +0.000, E1   +56.685, E3 +263400.508}
SPL {X  -158.009, Y  +328.771, Z    +0.000, E1   +56.325, E3 +263410.868}
SPL {X  -156.065, Y  +322.971, Z    +0.000, E1   +56.177, E3 +263419.212}
SPL {X  -154.487, Y  +318.719, Z    +0.000, E1   +55.733, E3 +263427.221}
SPL {X  -151.902, Y  +312.426, Z    +0.000, E1   +55.494, E3 +263436.696}
SPL {X  -149.742, Y  +307.668, Z    +0.000, E1   +54.896, E3 +263445.908}
SPL {X  -146.487, Y  +301.160, Z    +0.000, E1   +54.808, E3 +263454.771}
SPL {X  -133.590, Y  +280.553, Z    +0.000, E1   +59.642, E3 +263455.728}
SPL {X  -112.638, Y  +257.040, Z    +0.000, E1   +51.417, E3 +263559.111}
ENDSPLINE

SPLINE
SPL {X  -115.209, Y  +259.476, Z    +0.000, E1   +49.595, E3 +263592.381}
SPL {X  -147.344, Y  +302.806, Z    +0.000, E1   +40.158, E3 +263681.843}
SPL {X  -160.798, Y  +338.700, Z    +0.000, E1   +25.294, E3 +263681.325}
SPL {X  -163.893, Y  +354.439, Z    +0.000, E1   +16.805, E3 +263675.799}
SPL {X  -165.158, Y  +365.746, Z    +0.000, E1   +10.198, E3 +263673.742}
SPL {X  -165.639, Y  +376.620, Z    +0.000, E1    +3.186, E3 +263673.542}
SPL {X  -165.650, Y  +381.477, Z    +0.000, E1    -0.622, E3 +263672.353}
SPL {X  -165.650, Y  +384.861, Z    +0.000, E1    -4.465, E3 +263671.755}
SPL {X  -165.650, Y  +388.792, Z    +0.000, E1    -9.482, E3 +263671.071}
SPL {X  -165.650, Y  +393.970, Z    +0.000, E1   -17.146, E3 +263670.228}
SPL {X  -165.650, Y  +401.614, Z    +0.000, E1   -27.619, E3 +263670.883}
SPL {X  -165.650, Y  +418.105, Z    +0.000, E1   -49.413, E3 +263666.291}
SPL {X  -165.650, Y  +465.736, Z    +0.000, E1   -65.678, E3 +263680.033}
SPL {X  -165.650, Y  +519.483, Z    +0.000, E1   -68.357, E3 +263706.218}
SPL {X  -165.650, Y  +548.869, Z    +0.000, E1   -62.199, E3 +263761.911}
ENDSPLINE

SPLINE
SPL {X  -165.650, Y  +530.735, Z    +0.000, E1   -57.778, E3 +263770.334}
ENDSPLINE

SPLINE
SPL {X  -165.650, Y  +536.777, Z    +0.000, E1   -57.774, E3 +263778.211}
SPL {X  -165.650, Y  +545.905, Z    +0.000, E1   -57.853, E3 +263789.500}
SPL {X  -165.650, Y  +553.630, Z    +0.000, E1   -57.616, E3 +263800.949}
SPL {X  -165.650, Y  +563.473, Z    +0.000, E1   -57.690, E3 +263813.313}
SPL {X  -165.650, Y  +573.011, Z    +0.000, E1   -57.610, E3 +263826.104}
SPL {X  -165.650, Y  +581.530, Z    +0.000, E1   -57.678, E3 +263836.702}
SPL {X  -165.650, Y  +589.475, Z    +0.000, E1   -57.572, E3 +263847.689}
SPL {X  -165.650, Y  +599.695, Z    +0.000, E1   -57.964, E3 +263858.305}
SPL {X  -165.650, Y  +606.915, Z    +0.000, E1   -57.651, E3 +263869.662}
SPL {X  -165.650, Y  +614.927, Z    +0.000, E1   -57.517, E3 +263880.932}
SPL {X  -165.650, Y  +624.337, Z    +0.000, E1   -57.671, E3 +263892.158}
SPL {X  -165.650, Y  +634.236, Z    +0.000, E1   -57.671, E3 +263905.008}
SPL {X  -165.650, Y  +644.287, Z    +0.000, E1   -57.872, E3 +263916.574}
SPL {X  -165.650, Y  +650.480, Z    +0.000, E1   -57.669, E3 +263925.879}
SPL {X  -165.650, Y  +657.986, Z    +0.000, E1   -57.646, E3 +263935.771}
SPL {X  -165.650, Y  +667.585, Z    +0.000, E1   -57.803, E3 +263947.167}
SPL {X  -165.634, Y  +677.794, Z    +0.000, E1   -57.650, E3 +263961.469}
SPL {X  -165.167, Y  +688.139, Z    +0.000, E1   -57.463, E3 +263976.048}
SPL {X  -164.323, Y  +696.426, Z    +0.000, E1   -57.565, E3 +263986.035}
SPL {X  -163.313, Y  +703.224, Z    +0.000, E1   -57.403, E3 +263995.929}
SPL {X  -161.906, Y  +710.520, Z    +0.000, E1   -57.149, E3 +264006.880}
SPL {X  -160.577, Y  +716.182, Z    +0.000, E1   -56.676, E3 +264017.141}
SPL {X  -158.520, Y  +723.576, Z    +0.000, E1   -56.758, E3 +264026.186}
SPL {X  -156.858, Y  +728.749, Z    +0.000, E1   -56.333, E3 +264035.329}
SPL {X  -155.155, Y  +733.525, Z    +0.000, E1   -55.869, E3 +264044.105}
SPL {X  -153.442, Y  +737.914, Z    +0.000, E1   -55.562, E3 +264051.510}
SPL {X  -150.574, Y  +744.547, Z    +0.000, E1   -55.310, E3 +264061.492}
SPL {X  -147.713, Y  +750.471, Z    +0.000, E1   -54.514, E3 +264073.155}
SPL {X  -139.786, Y  +764.381, Z    +0.000, E1   -57.209, E3 +264077.343}
SPL {X  -110.324, Y  +799.066, Z    +0.000, E1   -54.396, E3 +264145.917}
SPL {X  -100.308, Y  +807.326, Z    +0.000, E1   -52.880, E3 +264190.485}
ENDSPLINE

SPLINE
SPL {X  -108.196, Y  +800.934, Z    +0.000, E1   -52.068, E3 +264282.811}
SPL {X  -147.753, Y  +750.393, Z    +0.000, E1   -39.863, E3 +264301.034}
SPL {X  -161.414, Y  +712.720, Z    +0.000, E1   -24.024, E3 +264300.376}
SPL {X  -164.278, Y  +696.774, Z    +0.000, E1   -15.225, E3 +264294.987}
SPL {X  -165.380, Y  +684.954, Z    +0.000, E1    -8.247, E3 +264297.770}
SPL {X  -165.650, Y  +675.104, Z    +0.000, E1    -1.512, E3 +264296.565}
SPL {X  -165.650, Y  +672.384, Z    +0.000, E1    +0.908, E3 +264295.455}
SPL {X  -165.650, Y  +669.968, Z    +0.000, E1    +3.584, E3 +264295.271}
SPL {X  -165.650, Y  +666.667, Z    +0.000, E1    +7.761, E3 +264294.950}
SPL {X  -165.650, Y  +662.028, Z    +0.000, E1   +14.359, E3 +264294.580}
SPL {X  -165.650, Y  +654.885, Z    +0.000, E1   +25.204, E3 +264293.095}
SPL {X  -165.650, Y  +641.882, Z    +0.000, E1   +46.566, E3 +264285.967}
SPL {X  -165.650, Y  +630.946, Z    +0.000, E1   +55.779, E3 +264286.641}
SPL {X  -165.650, Y  +590.135, Z    +0.000, E1   +59.110, E3 +264319.261}
SPL {X  -165.650, Y  +491.251, Z    +0.000, E1   +65.373, E3 +264378.690}
ENDSPLINE

SPLINE
SPL {X  -165.650, Y  +514.386, Z    +0.000, E1   +58.403, E3 +264402.240}
ENDSPLINE

SPLINE
SPL {X  -165.650, Y  +502.532, Z    +0.000, E1   +57.988, E3 +264419.856}
SPL {X  -165.650, Y  +493.307, Z    +0.000, E1   +58.045, E3 +264431.125}
SPL {X  -165.650, Y  +485.167, Z    +0.000, E1   +58.003, E3 +264441.903}
ENDSPLINE

SPLINE
SPL {X  -165.650, Y  +509.193, Z    +0.000, E1   +50.604, E3 +264452.870}
ENDSPLINE

SPLINE
SPL {X  -165.650, Y  +503.302, Z    +0.000, E1   +50.402, E3 +264463.966}
SPL {X  -165.650, Y  +495.166, Z    +0.000, E1   +51.070, E3 +264473.543}
SPL {X  -165.650, Y  +485.807, Z    +0.000, E1   +51.973, E3 +264483.276}
SPL {X  -165.650, Y  +478.030, Z    +0.000, E1   +52.389, E3 +264493.083}
SPL {X  -165.650, Y  +467.527, Z    +0.000, E1   +53.334, E3 +264503.577}
SPL {X  -165.650, Y  +457.379, Z    +0.000, E1   +53.935, E3 +264515.120}
SPL {X  -165.650, Y  +444.120, Z    +0.000, E1   +54.815, E3 +264529.166}
SPL {X  -165.650, Y  +431.771, Z    +0.000, E1   +55.549, E3 +264541.996}
SPL {X  -165.650, Y  +420.799, Z    +0.000, E1   +56.452, E3 +264551.382}
SPL {X  -165.650, Y  +406.746, Z    +0.000, E1   +57.489, E3 +264563.426}
SPL {X  -165.650, Y  +399.455, Z    +0.000, E1   +57.184, E3 +264574.848}
SPL {X  -165.650, Y  +388.492, Z    +0.000, E1   +57.709, E3 +264585.768}
SPL {X  -165.650, Y  +379.894, Z    +0.000, E1   +57.709, E3 +264596.871}
SPL {X  -165.399, Y  +369.388, Z    +0.000, E1   +57.657, E3 +264610.965}
SPL {X  -164.717, Y  +360.945, Z    +0.000, E1   +57.468, E3 +264622.903}
SPL {X  -163.867, Y  +354.258, Z    +0.000, E1   +57.359, E3 +264632.348}
SPL {X  -162.678, Y  +347.264, Z    +0.000, E1   +57.150, E3 +264642.689}
SPL {X  -161.618, Y  +342.173, Z    +0.000, E1   +56.783, E3 +264651.574}
SPL {X  -159.878, Y  +335.155, Z    +0.000, E1   +56.685, E3 +264661.378}
SPL {X  -158.009, Y  +328.771, Z    +0.000, E1   +56.325, E3 +264671.738}
SPL {X  -156.065, Y  +322.971, Z    +0.000, E1   +56.177, E3 +264680.082}
SPL {X  -154.487, Y  +318.719, Z    +0.000, E1   +55.733, E3 +264688.090}
SPL {X  -151.902, Y  +312.426, Z    +0.000, E1   +55.494, E3 +264697.565}
SPL {X  -149.742, Y  +307.668, Z    +0.000, E1   +54.896, E3 +264706.777}
SPL {X  -146.487, Y  +301.160, Z    +0.000, E1   +54.808, E3 +264715.640}
SPL {X  -133.590, Y  +280.553, Z    +0.000, E1   +59.642, E3 +264716.597}
SPL {X  -112.638, Y  +257.040, Z    +0.000, E1   +51.417, E3 +264819.980}
ENDSPLINE

SPLINE
SPL {X  -115.209, Y  +259.476, Z    +0.000, E1   +49.595, E3 +264853.251}
SPL {X  -147.344, Y  +302.806, Z    +0.000, E1   +40.158, E3 +264942.713}
SPL {X  -160.798, Y  +338.700, Z    +0.000, E1   +25.294, E3 +264942.195}
SPL {X  -163.893, Y  +354.439, Z    +0.000, E1   +16.805, E3 +264936.669}
SPL {X  -165.158, Y  +365.746, Z    +0.000, E1   +10.198, E3 +264934.612}
SPL {X  -165.639, Y  +376.620, Z    +0.000, E1    +3.186, E3 +264934.412}
SPL {X  -165.650, Y  +381.477, Z    +0.000, E1    -0.622, E3 +264933.222}
SPL {X  -165.650, Y  +386.363, Z    +0.000, E1    -6.162, E3 +264932.571}
SPL {X  -165.650, Y  +392.511, Z    +0.000, E1   -14.940, E3 +264931.011}
SPL {X  -165.650, Y  +398.939, Z    +0.000, E1   -23.851, E3 +264932.396}
SPL {X  -165.650, Y  +404.249, Z    +0.000, E1   -31.650, E3 +264931.117}
SPL {X  -165.650, Y  +418.105, Z    +0.000, E1   -49.413, E3 +264927.160}
SPL {X  -165.650, Y  +465.736, Z    +0.000, E1   -65.678, E3 +264940.903}
SPL {X  -165.650, Y  +519.483, Z    +0.000, E1   -68.357, E3 +264967.088}
SPL {X  -165.650, Y  +548.869, Z    +0.000, E1   -62.199, E3 +265022.780}
ENDSPLINE

SPLINE
SPL {X  -165.650, Y  +530.735, Z    +0.000, E1   -57.778, E3 +265031.204}
ENDSPLINE

SPLINE
SPL {X  -165.650, Y  +536.777, Z    +0.000, E1   -57.774, E3 +265039.081}
SPL {X  -165.650, Y  +545.905, Z    +0.000, E1   -57.853, E3 +265050.369}
SPL {X  -165.650, Y  +553.630, Z    +0.000, E1   -57.616, E3 +265061.819}
SPL {X  -165.650, Y  +563.473, Z    +0.000, E1   -57.690, E3 +265074.183}
SPL {X  -165.650, Y  +573.011, Z    +0.000, E1   -57.610, E3 +265086.974}
SPL {X  -165.650, Y  +581.530, Z    +0.000, E1   -57.678, E3 +265097.572}
SPL {X  -165.650, Y  +589.475, Z    +0.000, E1   -57.572, E3 +265108.559}
SPL {X  -165.650, Y  +599.695, Z    +0.000, E1   -57.964, E3 +265119.175}
SPL {X  -165.650, Y  +606.915, Z    +0.000, E1   -57.651, E3 +265130.532}
SPL {X  -165.650, Y  +614.927, Z    +0.000, E1   -57.517, E3 +265141.801}
SPL {X  -165.650, Y  +624.337, Z    +0.000, E1   -57.671, E3 +265153.027}
SPL {X  -165.650, Y  +634.236, Z    +0.000, E1   -57.671, E3 +265165.878}
SPL {X  -165.650, Y  +647.519, Z    +0.000, E1   -57.817, E3 +265182.205}
SPL {X  -165.650, Y  +657.986, Z    +0.000, E1   -57.646, E3 +265196.641}
SPL {X  -165.650, Y  +667.585, Z    +0.000, E1   -57.803, E3 +265208.036}
SPL {X  -165.634, Y  +677.794, Z    +0.000, E1   -57.650, E3 +265222.339}
SPL {X  -165.167, Y  +688.139, Z    +0.000, E1   -57.463, E3 +265236.918}
SPL {X  -164.323, Y  +696.426, Z    +0.000, E1   -57.565, E3 +265246.905}
SPL {X  -163.313, Y  +703.224, Z    +0.000, E1   -57.403, E3 +265256.799}
SPL {X  -161.906, Y  +710.520, Z    +0.000, E1   -57.149, E3 +265267.750}
SPL {X  -160.577, Y  +716.182, Z    +0.000, E1   -56.676, E3 +265278.011}
SPL {X  -158.520, Y  +723.576, Z    +0.000, E1   -56.758, E3 +265287.056}
SPL {X  -156.858, Y  +728.749, Z    +0.000, E1   -56.333, E3 +265296.198}
SPL {X  -155.155, Y  +733.525, Z    +0.000, E1   -55.869, E3 +265304.975}
SPL {X  -153.442, Y  +737.914, Z    +0.000, E1   -55.562, E3 +265312.379}
SPL {X  -150.574, Y  +744.547, Z    +0.000, E1   -55.310, E3 +265322.362}
SPL {X  -147.713, Y  +750.471, Z    +0.000, E1   -54.514, E3 +265334.025}
SPL {X  -139.786, Y  +764.381, Z    +0.000, E1   -57.209, E3 +265338.213}
SPL {X  -110.324, Y  +799.066, Z    +0.000, E1   -54.396, E3 +265406.787}
SPL {X  -100.308, Y  +807.326, Z    +0.000, E1   -52.880, E3 +265451.354}
ENDSPLINE

SPLINE
SPL {X  -108.196, Y  +800.934, Z    +0.000, E1   -52.068, E3 +265543.681}
SPL {X  -144.673, Y  +756.182, Z    +0.000, E1   -41.752, E3 +265561.759}
SPL {X  -160.601, Y  +716.087, Z    +0.000, E1   -25.730, E3 +265561.387}
SPL {X  -164.850, Y  +691.761, Z    +0.000, E1   -12.424, E3 +265558.655}
SPL {X  -165.596, Y  +679.730, Z    +0.000, E1    -4.777, E3 +265557.528}
SPL {X  -165.650, Y  +674.376, Z    +0.000, E1    -0.866, E3 +265557.443}
SPL {X  -165.650, Y  +672.384, Z    +0.000, E1    +0.908, E3 +265556.324}
SPL {X  -165.650, Y  +669.093, Z    +0.000, E1    +4.549, E3 +265556.176}
SPL {X  -165.650, Y  +663.273, Z    +0.000, E1   +12.448, E3 +265555.413}
SPL {X  -165.650, Y  +654.885, Z    +0.000, E1   +25.204, E3 +265553.965}
SPL {X  -165.650, Y  +641.882, Z    +0.000, E1   +46.566, E3 +265546.836}
SPL {X  -165.650, Y  +630.946, Z    +0.000, E1   +55.779, E3 +265547.511}
SPL {X  -165.650, Y  +590.135, Z    +0.000, E1   +59.110, E3 +265580.130}
SPL {X  -165.650, Y  +491.251, Z    +0.000, E1   +65.373, E3 +265639.560}
ENDSPLINE

SPLINE
SPL {X  -165.650, Y  +517.534, Z    +0.000, E1   +59.090, E3 +265654.157}
ENDSPLINE

SPLINE
SPL {X  -165.650, Y  +515.821, Z    +0.000, E1   +58.153, E3 +265662.605}
SPL {X  -165.650, Y  +506.715, Z    +0.000, E1   +58.090, E3 +265674.693}
SPL {X  -165.650, Y  +496.085, Z    +0.000, E1   +57.984, E3 +265688.941}
SPL {X  -165.650, Y  +485.167, Z    +0.000, E1   +58.003, E3 +265702.772}
ENDSPLINE

SPLINE
SPL {X  -165.650, Y  +505.180, Z    +0.000, E1   +52.333, E3 +265709.525}
SPL {X  -165.650, Y  +506.534, Z    +0.000, E1   +50.148, E3 +265720.984}
ENDSPLINE

SPLINE
SPL {X  -165.650, Y  +495.166, Z    +0.000, E1   +51.070, E3 +265734.413}
SPL {X  -165.650, Y  +485.807, Z    +0.000, E1   +51.973, E3 +265744.145}
SPL {X  -165.650, Y  +478.030, Z    +0.000, E1   +52.389, E3 +265753.952}
SPL {X  -165.650, Y  +467.527, Z    +0.000, E1   +53.334, E3 +265764.446}
SPL {X  -165.650, Y  +453.744, Z    +0.000, E1   +54.190, E3 +265779.927}
SPL {X  -165.650, Y  +440.843, Z    +0.000, E1   +55.023, E3 +265793.348}
SPL {X  -165.650, Y  +431.771, Z    +0.000, E1   +55.549, E3 +265802.865}
SPL {X  -165.650, Y  +420.799, Z    +0.000, E1   +56.452, E3 +265812.251}
SPL {X  -165.650, Y  +409.731, Z    +0.000, E1   +57.273, E3 +265821.739}
SPL {X  -165.650, Y  +399.687, Z    +0.000, E1   +57.433, E3 +265833.924}
SPL {X  -165.650, Y  +388.492, Z    +0.000, E1   +57.709, E3 +265846.637}
SPL {X  -165.650, Y  +379.894, Z    +0.000, E1   +57.709, E3 +265857.741}
SPL {X  -165.399, Y  +369.388, Z    +0.000, E1   +57.657, E3 +265871.835}
SPL {X  -164.717, Y  +360.945, Z    +0.000, E1   +57.468, E3 +265883.773}
SPL {X  -163.867, Y  +354.258, Z    +0.000, E1   +57.359, E3 +265893.217}
SPL {X  -162.678, Y  +347.264, Z    +0.000, E1   +57.150, E3 +265903.558}
SPL {X  -161.618, Y  +342.173, Z    +0.000, E1   +56.783, E3 +265912.444}
SPL {X  -159.878, Y  +335.155, Z    +0.000, E1   +56.685, E3 +265922.248}
SPL {X  -158.009, Y  +328.771, Z    +0.000, E1   +56.325, E3 +265932.607}
SPL {X  -156.065, Y  +322.971, Z    +0.000, E1   +56.177, E3 +265940.951}
SPL {X  -153.731, Y  +316.803, Z    +0.000, E1   +55.737, E3 +265951.528}
SPL {X  -150.320, Y  +308.902, Z    +0.000, E1   +55.085, E3 +265965.224}
SPL {X  -147.957, Y  +304.011, Z    +0.000, E1   +54.431, E3 +265974.686}
SPL {X  -144.791, Y  +298.030, Z    +0.000, E1   +55.214, E3 +265978.544}
SPL {X  -133.590, Y  +280.553, Z    +0.000, E1   +59.642, E3 +265977.467}
SPL {X  -112.638, Y  +257.040, Z    +0.000, E1   +51.417, E3 +266080.850}
ENDSPLINE

SPLINE
SPL {X  -115.209, Y  +259.476, Z    +0.000, E1   +49.595, E3 +266114.120}
SPL {X  -147.344, Y  +302.806, Z    +0.000, E1   +40.158, E3 +266203.582}
SPL {X  -160.798, Y  +338.700, Z    +0.000, E1   +25.294, E3 +266203.064}
SPL {X  -163.893, Y  +354.439, Z    +0.000, E1   +16.805, E3 +266197.538}
SPL {X  -165.158, Y  +365.746, Z    +0.000, E1   +10.198, E3 +266195.481}
SPL {X  -165.580, Y  +373.688, Z    +0.000, E1    +5.094, E3 +266195.218}
SPL {X  -165.650, Y  +379.719, Z    +0.000, E1    +0.894, E3 +266194.648}
SPL {X  -165.650, Y  +383.454, Z    +0.000, E1    -2.667, E3 +266193.716}
SPL {X  -165.650, Y  +387.779, Z    +0.000, E1    -8.159, E3 +266193.390}
SPL {X  -165.650, Y  +392.511, Z    +0.000, E1   -14.940, E3 +266191.880}
SPL {X  -165.650, Y  +401.614, Z    +0.000, E1   -27.619, E3 +266192.622}
SPL {X  -165.650, Y  +418.105, Z    +0.000, E1   -49.413, E3 +266188.030}
SPL {X  -165.650, Y  +465.736, Z    +0.000, E1   -65.678, E3 +266201.772}
SPL {X  -165.650, Y  +519.483, Z    +0.000, E1   -68.357, E3 +266227.957}
SPL {X  -165.650, Y  +548.869, Z    +0.000, E1   -62.199, E3 +266283.650}
ENDSPLINE

SPLINE
SPL {X  -165.650, Y  +534.780, Z    +0.000, E1   -57.803, E3 +266297.299}
ENDSPLINE

SPLINE
SPL {X  -165.650, Y  +545.905, Z    +0.000, E1   -57.853, E3 +266311.239}
SPL {X  -165.650, Y  +555.746, Z    +0.000, E1   -57.571, E3 +266325.876}
SPL {X  -165.650, Y  +566.557, Z    +0.000, E1   -57.834, E3 +266338.004}
SPL {X  -165.650, Y  +573.011, Z    +0.000, E1   -57.610, E3 +266347.843}
SPL {X  -165.650, Y  +581.530, Z    +0.000, E1   -57.678, E3 +266358.442}
SPL {X  -165.650, Y  +589.475, Z    +0.000, E1   -57.572, E3 +266369.428}
SPL {X  -165.650, Y  +599.695, Z    +0.000, E1   -57.964, E3 +266380.045}
SPL {X  -165.650, Y  +606.915, Z    +0.000, E1   -57.651, E3 +266391.401}
SPL {X  -165.650, Y  +614.927, Z    +0.000, E1   -57.517, E3 +266402.671}
SPL {X  -165.650, Y  +624.337, Z    +0.000, E1   -57.671, E3 +266413.897}
SPL {X  -165.650, Y  +634.236, Z    +0.000, E1   -57.671, E3 +266426.747}
SPL {X  -165.650, Y  +647.519, Z    +0.000, E1   -57.817, E3 +266443.075}
SPL {X  -165.650, Y  +657.986, Z    +0.000, E1   -57.646, E3 +266457.510}
SPL {X  -165.650, Y  +667.585, Z    +0.000, E1   -57.803, E3 +266468.906}
SPL {X  -165.634, Y  +677.794, Z    +0.000, E1   -57.650, E3 +266483.208}
SPL {X  -165.167, Y  +688.139, Z    +0.000, E1   -57.463, E3 +266497.788}
SPL {X  -164.009, Y  +698.761, Z    +0.000, E1   -57.613, E3 +266510.561}
SPL {X  -162.382, Y  +708.242, Z    +0.000, E1   -57.205, E3 +266525.487}
SPL {X  -160.577, Y  +716.182, Z    +0.000, E1   -56.676, E3 +266538.880}
SPL {X  -158.520, Y  +723.576, Z    +0.000, E1   -56.758, E3 +266547.925}
SPL {X  -156.858, Y  +728.749, Z    +0.000, E1   -56.333, E3 +266557.068}
SPL {X  -155.155, Y  +733.525, Z    +0.000, E1   -55.869, E3 +266565.844}
SPL {X  -152.530, Y  +740.111, Z    +0.000, E1   -55.545, E3 +266576.321}
SPL {X  -149.838, Y  +746.130, Z    +0.000, E1   -55.135, E3 +266586.041}
SPL {X  -147.713, Y  +750.471, Z    +0.000, E1   -54.514, E3 +266594.894}
SPL {X  -139.786, Y  +764.381, Z    +0.000, E1   -57.209, E3 +266599.082}
SPL {X  -110.324, Y  +799.066, Z    +0.000, E1   -54.396, E3 +266667.656}
SPL {X  -100.308, Y  +807.326, Z    +0.000, E1   -52.880, E3 +266712.224}
ENDSPLINE

SPLINE
SPL {X  -108.196, Y  +800.934, Z    +0.000, E1   -52.068, E3 +266804.550}
SPL {X  -147.753, Y  +750.393, Z    +0.000, E1   -39.863, E3 +266822.773}
SPL {X  -161.414, Y  +712.720, Z    +0.000, E1   -24.024, E3 +266822.115}
SPL {X  -164.278, Y  +696.774, Z    +0.000, E1   -15.225, E3 +266816.727}
SPL {X  -165.078, Y  +689.251, Z    +0.000, E1   -10.876, E3 +266820.879}
SPL {X  -165.596, Y  +679.730, Z    +0.000, E1    -4.777, E3 +266818.398}
SPL {X  -165.650, Y  +674.376, Z    +0.000, E1    -0.866, E3 +266818.313}
SPL {X  -165.650, Y  +672.384, Z    +0.000, E1    +0.908, E3 +266817.194}
SPL {X  -165.650, Y  +669.093, Z    +0.000, E1    +4.549, E3 +266817.046}
SPL {X  -165.650, Y  +663.273, Z    +0.000, E1   +12.448, E3 +266816.283}
SPL {X  -165.650, Y  +657.199, Z    +0.000, E1   +21.720, E3 +266815.552}
SPL {X  -165.650, Y  +652.963, Z    +0.000, E1   +28.395, E3 +266814.237}
SPL {X  -165.650, Y  +641.882, Z    +0.000, E1   +46.566, E3 +266807.706}
SPL {X  -165.650, Y  +630.946, Z    +0.000, E1   +55.779, E3 +266808.380}
SPL {X  -165.650, Y  +590.135, Z    +0.000, E1   +59.110, E3 +266841.000}
SPL {X  -165.650, Y  +491.251, Z    +0.000, E1   +65.373, E3 +266900.429}
ENDSPLINE

SPLINE
SPL {X  -165.650, Y  +516.236, Z    +0.000, E1   +58.457, E3 +266921.110}
ENDSPLINE

SPLINE
SPL {X  -165.650, Y  +506.715, Z    +0.000, E1   +58.090, E3 +266935.563}
SPL {X  -165.650, Y  +496.085, Z    +0.000, E1   +57.984, E3 +266949.810}
SPL {X  -165.650, Y  +485.167, Z    +0.000, E1   +58.003, E3 +266963.642}
ENDSPLINE

SPLINE
SPL {X  -165.650, Y  +505.180, Z    +0.000, E1   +52.333, E3 +266970.394}
SPL {X  -165.650, Y  +506.534, Z    +0.000, E1   +50.148, E3 +266981.854}
ENDSPLINE

SPLINE
SPL {X  -165.650, Y  +495.166, Z    +0.000, E1   +51.070, E3 +266995.282}
SPL {X  -165.650, Y  +485.807, Z    +0.000, E1   +51.973, E3 +267005.015}
SPL {X  -165.650, Y  +475.672, Z    +0.000, E1   +52.573, E3 +267017.469}
SPL {X  -165.650, Y  +459.814, Z    +0.000, E1   +53.888, E3 +267033.658}
SPL {X  -165.650, Y  +448.876, Z    +0.000, E1   +54.452, E3 +267046.153}
SPL {X  -165.650, Y  +440.843, Z    +0.000, E1   +55.023, E3 +267054.217}
SPL {X  -165.650, Y  +431.771, Z    +0.000, E1   +55.549, E3 +267063.735}
SPL {X  -165.650, Y  +420.799, Z    +0.000, E1   +56.452, E3 +267073.121}
SPL {X  -165.650, Y  +406.746, Z    +0.000, E1   +57.489, E3 +267085.165}
SPL {X  -165.650, Y  +399.455, Z    +0.000, E1   +57.184, E3 +267096.587}
SPL {X  -165.650, Y  +388.492, Z    +0.000, E1   +57.709, E3 +267107.507}
SPL {X  -165.650, Y  +379.894, Z    +0.000, E1   +57.709, E3 +267118.610}
SPL {X  -165.399, Y  +369.388, Z    +0.000, E1   +57.657, E3 +267132.704}
SPL {X  -164.717, Y  +360.945, Z    +0.000, E1   +57.468, E3 +267144.642}
SPL {X  -163.867, Y  +354.258, Z    +0.000, E1   +57.359, E3 +267154.087}
SPL {X  -162.678, Y  +347.264, Z    +0.000, E1   +57.150, E3 +267164.428}
SPL {X  -160.825, Y  +338.812, Z    +0.000, E1   +56.892, E3 +267177.170}
SPL {X  -158.481, Y  +330.294, Z    +0.000, E1   +56.303, E3 +267191.688}
SPL {X  -156.065, Y  +322.971, Z    +0.000, E1   +56.177, E3 +267201.821}
SPL {X  -154.487, Y  +318.719, Z    +0.000, E1   +55.733, E3 +267209.829}
SPL {X  -151.902, Y  +312.426, Z    +0.000, E1   +55.494, E3 +267219.304}
SPL {X  -148.935, Y  +305.985, Z    +0.000, E1   +54.737, E3 +267231.681}
SPL {X  -144.791, Y  +298.030, Z    +0.000, E1   +55.214, E3 +267239.414}
SPL {X  -133.590, Y  +280.553, Z    +0.000, E1   +59.642, E3 +267238.336}
SPL {X  -112.638, Y  +257.040, Z    +0.000, E1   +51.417, E3 +267341.719}
ENDSPLINE

